LIN {X 104.168,Y 46.841,Z 66.500,A 180.000,B 0.000,C 180.000} C_DIS
LIN {X 104.160,Y 46.662,Z 66.500,A 180.000,B 0.000,C 180.000} C_DIS
LIN {X 104.143,Y 46.483,Z 66.500,A 180.000,B 0.000,C 180.000} C_DIS
LIN {X 104.121,Y 46.275,Z 66.500,A 180.000,B 0.000,C 180.000} C_DIS
LIN {X 104.105,Y 46.126,Z 66.500,A 180.000,B 0.000,C 180.000} C_DIS
LIN {X 104.086,Y 45.947,Z 66.500,A 180.000,B 0.000,C 180.000} C_DIS
LIN {X 104.059,Y 45.768,Z 66.500,A 180.000,B 0.000,C 180.000} C_DIS
LIN {X 103.998,Y 45.411,Z 66.500,A 180.000,B 0.000,C 180.000} C_DIS
LIN {X 103.967,Y 45.232,Z 66.500,A 180.000,B 0.000,C 180.000} C_DIS
LIN {X 103.929,Y 45.053,Z 66.500,A 180.000,B 0.000,C 180.000} C_DIS
LIN {X 103.845,Y 44.696,Z 66.500,A 180.000,B 0.000,C 180.000} C_DIS
LIN {X 103.802,Y 44.517,Z 66.500,A 180.000,B 0.000,C 180.000} C_DIS
LIN {X 103.752,Y 44.338,Z 66.500,A 180.000,B 0.000,C 180.000} C_DIS
LIN {X 103.644,Y 43.981,Z 66.500,A 180.000,B 0.000,C 180.000} C_DIS
LIN {X 103.589,Y 43.802,Z 66.500,A 180.000,B 0.000,C 180.000} C_DIS
LIN {X 103.526,Y 43.623,Z 66.500,A 180.000,B 0.000,C 180.000} C_DIS
LIN {X 103.392,Y 43.266,Z 66.500,A 180.000,B 0.000,C 180.000} C_DIS
LIN {X 103.332,Y 43.106,Z 66.500,A 180.000,B 0.000,C 180.000} C_DIS
LIN {X 103.325,Y 43.087,Z 66.500,A 180.000,B 0.000,C 180.000} C_DIS
LIN {X 103.247,Y 42.908,Z 66.500,A 180.000,B 0.000,C 180.000} C_DIS
LIN {X 103.087,Y 42.550,Z 66.500,A 180.000,B 0.000,C 180.000} C_DIS
LIN {X 103.005,Y 42.372,Z 66.500,A 180.000,B 0.000,C 180.000} C_DIS
LIN {X 102.975,Y 42.314,Z 66.500,A 180.000,B 0.000,C 180.000} C_DIS
LIN {X 102.724,Y 41.835,Z 66.500,A 180.000,B 0.000,C 180.000} C_DIS
LIN {X 102.623,Y 41.657,Z 66.500,A 180.000,B 0.000,C 180.000} C_DIS
LIN {X 102.406,Y 41.299,Z 66.500,A 180.000,B 0.000,C 180.000} C_DIS
LIN {X 102.296,Y 41.120,Z 66.500,A 180.000,B 0.000,C 180.000} C_DIS
LIN {X 102.260,Y 41.067,Z 66.500,A 180.000,B 0.000,C 180.000} C_DIS
LIN {X 102.172,Y 40.942,Z 66.500,A 180.000,B 0.000,C 180.000} C_DIS
LIN {X 101.923,Y 40.584,Z 66.500,A 180.000,B 0.000,C 180.000} C_DIS
LIN {X 101.902,Y 40.554,Z 66.500,A 180.000,B 0.000,C 180.000} C_DIS
LIN {X 101.788,Y 40.405,Z 66.500,A 180.000,B 0.000,C 180.000} C_DIS
LIN {X 101.504,Y 40.048,Z 66.500,A 180.000,B 0.000,C 180.000} C_DIS
LIN {X 101.366,Y 39.883,Z 66.500,A 180.000,B 0.000,C 180.000} C_DIS
LIN {X 101.008,Y 39.486,Z 66.500,A 180.000,B 0.000,C 180.000} C_DIS
LIN {X 100.861,Y 39.333,Z 66.500,A 180.000,B 0.000,C 180.000} C_DIS
LIN {X 100.472,Y 38.952,Z 66.500,A 180.000,B 0.000,C 180.000} C_DIS
LIN {X 100.300,Y 38.796,Z 66.500,A 180.000,B 0.000,C 180.000} C_DIS
LIN {X 99.936,Y 38.482,Z 66.500,A 180.000,B 0.000,C 180.000} C_DIS
LIN {X 99.885,Y 38.439,Z 66.500,A 180.000,B 0.000,C 180.000} C_DIS
LIN {X 99.757,Y 38.338,Z 66.500,A 180.000,B 0.000,C 180.000} C_DIS
LIN {X 99.399,Y 38.067,Z 66.500,A 180.000,B 0.000,C 180.000} C_DIS
LIN {X 99.221,Y 37.936,Z 66.500,A 180.000,B 0.000,C 180.000} C_DIS
LIN {X 99.171,Y 37.902,Z 66.500,A 180.000,B 0.000,C 180.000} C_DIS
LIN {X 98.863,Y 37.698,Z 66.500,A 180.000,B 0.000,C 180.000} C_DIS
LIN {X 98.684,Y 37.580,Z 66.500,A 180.000,B 0.000,C 180.000} C_DIS
LIN {X 98.627,Y 37.545,Z 66.500,A 180.000,B 0.000,C 180.000} C_DIS
LIN {X 98.505,Y 37.474,Z 66.500,A 180.000,B 0.000,C 180.000} C_DIS
LIN {X 98.148,Y 37.268,Z 66.500,A 180.000,B 0.000,C 180.000} C_DIS
LIN {X 98.005,Y 37.187,Z 66.500,A 180.000,B 0.000,C 180.000} C_DIS
LIN {X 97.969,Y 37.169,Z 66.500,A 180.000,B 0.000,C 180.000} C_DIS
LIN {X 97.790,Y 37.080,Z 66.500,A 180.000,B 0.000,C 180.000} C_DIS
LIN {X 97.433,Y 36.903,Z 66.500,A 180.000,B 0.000,C 180.000} C_DIS
LIN {X 97.272,Y 36.830,Z 66.500,A 180.000,B 0.000,C 180.000} C_DIS
LIN {X 96.846,Y 36.651,Z 66.500,A 180.000,B 0.000,C 180.000} C_DIS
LIN {X 96.718,Y 36.598,Z 66.500,A 180.000,B 0.000,C 180.000} C_DIS
LIN {X 96.539,Y 36.533,Z 66.500,A 180.000,B 0.000,C 180.000} C_DIS
LIN {X 96.181,Y 36.409,Z 66.500,A 180.000,B 0.000,C 180.000} C_DIS
LIN {X 96.003,Y 36.347,Z 66.500,A 180.000,B 0.000,C 180.000} C_DIS
LIN {X 95.824,Y 36.296,Z 66.500,A 180.000,B 0.000,C 180.000} C_DIS
LIN {X 95.466,Y 36.196,Z 66.500,A 180.000,B 0.000,C 180.000} C_DIS
LIN {X 95.288,Y 36.147,Z 66.500,A 180.000,B 0.000,C 180.000} C_DIS
LIN {X 95.141,Y 36.115,Z 66.500,A 180.000,B 0.000,C 180.000} C_DIS
LIN {X 94.751,Y 36.032,Z 66.500,A 180.000,B 0.000,C 180.000} C_DIS
LIN {X 94.573,Y 35.995,Z 66.500,A 180.000,B 0.000,C 180.000} C_DIS
LIN {X 94.394,Y 35.967,Z 66.500,A 180.000,B 0.000,C 180.000} C_DIS
LIN {X 94.036,Y 35.915,Z 66.500,A 180.000,B 0.000,C 180.000} C_DIS
LIN {X 93.857,Y 35.889,Z 66.500,A 180.000,B 0.000,C 180.000} C_DIS
LIN {X 93.679,Y 35.872,Z 66.500,A 180.000,B 0.000,C 180.000} C_DIS
LIN {X 93.321,Y 35.843,Z 66.500,A 180.000,B 0.000,C 180.000} C_DIS
LIN {X 93.142,Y 35.828,Z 66.500,A 180.000,B 0.000,C 180.000} C_DIS
LIN {X 92.964,Y 35.822,Z 66.500,A 180.000,B 0.000,C 180.000} C_DIS
LIN {X 92.606,Y 35.814,Z 66.500,A 180.000,B 0.000,C 180.000} C_DIS
LIN {X 92.427,Y 35.811,Z 66.500,A 180.000,B 0.000,C 180.000} C_DIS
LIN {X 92.249,Y 35.815,Z 66.500,A 180.000,B 0.000,C 180.000} C_DIS
LIN {X 91.712,Y 35.838,Z 66.500,A 180.000,B 0.000,C 180.000} C_DIS
LIN {X 91.533,Y 35.852,Z 66.500,A 180.000,B 0.000,C 180.000} C_DIS
LIN {X 90.997,Y 35.908,Z 66.500,A 180.000,B 0.000,C 180.000} C_DIS
LIN {X 90.872,Y 35.926,Z 66.500,A 180.000,B 0.000,C 180.000} C_DIS
; Link Move Starts
LIN {X 90.783,Y 35.936,Z 66.500,A 180.000,B 0.000,C 180.000} C_DIS
LIN {X 90.702,Y 35.950,Z 66.500,A 180.000,B 0.000,C 180.000} C_DIS
LIN {X 90.699,Y 35.950,Z 66.500,A 180.000,B 0.000,C 180.000} C_DIS
LIN {X 90.693,Y 35.947,Z 66.500,A 180.000,B 0.000,C 180.000} C_DIS
LIN {X 90.541,Y 35.852,Z 66.500,A 180.000,B 0.000,C 180.000} C_DIS
LIN {X 90.371,Y 35.764,Z 66.499,A 180.000,B 0.000,C 180.000} C_DIS
LIN {X 90.194,Y 35.689,Z 66.499,A 180.000,B 0.000,C 180.000} C_DIS
LIN {X 90.035,Y 35.634,Z 66.498,A 180.000,B 0.000,C 180.000} C_DIS
LIN {X 89.873,Y 35.590,Z 66.497,A 180.000,B 0.000,C 180.000} C_DIS
LIN {X 89.718,Y 35.559,Z 66.496,A 180.000,B 0.000,C 180.000} C_DIS
LIN {X 89.562,Y 35.538,Z 66.495,A 180.000,B 0.000,C 180.000} C_DIS
LIN {X 89.405,Y 35.527,Z 66.494,A 180.000,B 0.000,C 180.000} C_DIS
LIN {X 89.247,Y 35.525,Z 66.493,A 180.000,B 0.000,C 180.000} C_DIS
LIN {X 89.090,Y 35.534,Z 66.492,A 180.000,B 0.000,C 180.000} C_DIS
LIN {X 88.934,Y 35.552,Z 66.490,A 180.000,B 0.000,C 180.000} C_DIS
LIN {X 88.779,Y 35.580,Z 66.489,A 180.000,B 0.000,C 180.000} C_DIS
LIN {X 88.626,Y 35.618,Z 66.487,A 180.000,B 0.000,C 180.000} C_DIS
LIN {X 88.326,Y 35.716,Z 66.483,A 180.000,B 0.000,C 180.000} C_DIS
LIN {X 88.028,Y 35.817,Z 66.479,A 180.000,B 0.000,C 180.000} C_DIS
LIN {X 87.730,Y 35.917,Z 66.475,A 180.000,B 0.000,C 180.000} C_DIS
LIN {X 87.431,Y 36.018,Z 66.470,A 180.000,B 0.000,C 180.000} C_DIS
LIN {X 87.282,Y 36.068,Z 66.467,A 180.000,B 0.000,C 180.000} C_DIS
LIN {X 87.133,Y 36.119,Z 66.465,A 180.000,B 0.000,C 180.000} C_DIS
LIN {X 86.983,Y 36.169,Z 66.462,A 180.000,B 0.000,C 180.000} C_DIS
LIN {X 86.834,Y 36.219,Z 66.459,A 180.000,B 0.000,C 180.000} C_DIS
LIN {X 86.685,Y 36.270,Z 66.456,A 180.000,B 0.000,C 180.000} C_DIS
LIN {X 86.536,Y 36.320,Z 66.453,A 180.000,B 0.000,C 180.000} C_DIS
LIN {X 86.386,Y 36.370,Z 66.450,A 180.000,B 0.000,C 180.000} C_DIS
LIN {X 86.237,Y 36.421,Z 66.446,A 180.000,B 0.000,C 180.000} C_DIS
LIN {X 86.088,Y 36.471,Z 66.443,A 180.000,B 0.000,C 180.000} C_DIS
LIN {X 85.939,Y 36.521,Z 66.440,A 180.000,B 0.000,C 180.000} C_DIS
LIN {X 85.789,Y 36.572,Z 66.436,A 180.000,B 0.000,C 180.000} C_DIS
LIN {X 85.640,Y 36.622,Z 66.433,A 180.000,B 0.000,C 180.000} C_DIS
LIN {X 85.491,Y 36.672,Z 66.429,A 180.000,B 0.000,C 180.000} C_DIS
LIN {X 85.342,Y 36.723,Z 66.425,A 180.000,B 0.000,C 180.000} C_DIS
LIN {X 85.193,Y 36.773,Z 66.421,A 180.000,B 0.000,C 180.000} C_DIS
LIN {X 85.043,Y 36.823,Z 66.417,A 180.000,B 0.000,C 180.000} C_DIS
LIN {X 84.894,Y 36.874,Z 66.413,A 180.000,B 0.000,C 180.000} C_DIS
LIN {X 84.745,Y 36.924,Z 66.409,A 180.000,B 0.000,C 180.000} C_DIS
LIN {X 84.596,Y 36.974,Z 66.405,A 180.000,B 0.000,C 180.000} C_DIS
LIN {X 84.446,Y 37.025,Z 66.401,A 180.000,B 0.000,C 180.000} C_DIS
LIN {X 84.297,Y 37.075,Z 66.397,A 180.000,B 0.000,C 180.000} C_DIS
LIN {X 84.148,Y 37.125,Z 66.392,A 180.000,B 0.000,C 180.000} C_DIS
LIN {X 83.999,Y 37.176,Z 66.388,A 180.000,B 0.000,C 180.000} C_DIS
LIN {X 83.849,Y 37.226,Z 66.383,A 180.000,B 0.000,C 180.000} C_DIS
LIN {X 83.700,Y 37.277,Z 66.379,A 180.000,B 0.000,C 180.000} C_DIS
LIN {X 83.551,Y 37.327,Z 66.374,A 180.000,B 0.000,C 180.000} C_DIS
LIN {X 83.402,Y 37.377,Z 66.369,A 180.000,B 0.000,C 180.000} C_DIS
LIN {X 83.252,Y 37.428,Z 66.364,A 180.000,B 0.000,C 180.000} C_DIS
LIN {X 83.103,Y 37.478,Z 66.359,A 180.000,B 0.000,C 180.000} C_DIS
LIN {X 82.954,Y 37.528,Z 66.355,A 180.000,B 0.000,C 180.000} C_DIS
LIN {X 82.879,Y 37.553,Z 66.352,A 180.000,B 0.000,C 180.000} C_DIS
LIN {X 82.805,Y 37.579,Z 66.350,A 180.000,B 0.000,C 180.000} C_DIS
LIN {X 82.730,Y 37.604,Z 66.347,A 180.000,B 0.000,C 180.000} C_DIS
LIN {X 82.655,Y 37.629,Z 66.344,A 180.000,B 0.000,C 180.000} C_DIS
LIN {X 82.581,Y 37.654,Z 66.342,A 180.000,B 0.000,C 180.000} C_DIS
LIN {X 82.506,Y 37.679,Z 66.339,A 180.000,B 0.000,C 180.000} C_DIS
LIN {X 82.432,Y 37.704,Z 66.337,A 180.000,B 0.000,C 180.000} C_DIS
LIN {X 82.282,Y 37.755,Z 66.332,A 180.000,B 0.000,C 180.000} C_DIS
LIN {X 82.133,Y 37.805,Z 66.326,A 180.000,B 0.000,C 180.000} C_DIS
LIN {X 81.984,Y 37.855,Z 66.321,A 180.000,B 0.000,C 180.000} C_DIS
LIN {X 81.835,Y 37.906,Z 66.315,A 180.000,B 0.000,C 180.000} C_DIS
LIN {X 81.685,Y 37.956,Z 66.310,A 180.000,B 0.000,C 180.000} C_DIS
LIN {X 81.536,Y 38.007,Z 66.305,A 180.000,B 0.000,C 180.000} C_DIS
LIN {X 81.462,Y 38.032,Z 66.302,A 180.000,B 0.000,C 180.000} C_DIS
LIN {X 81.312,Y 38.082,Z 66.296,A 180.000,B 0.000,C 180.000} C_DIS
LIN {X 81.089,Y 38.158,Z 66.288,A 180.000,B 0.000,C 180.000} C_DIS
LIN {X 80.939,Y 38.208,Z 66.283,A 180.000,B 0.000,C 180.000} C_DIS
LIN {X 80.865,Y 38.233,Z 66.280,A 180.000,B 0.000,C 180.000} C_DIS
LIN {X 80.715,Y 38.283,Z 66.274,A 180.000,B 0.000,C 180.000} C_DIS
LIN {X 80.492,Y 38.359,Z 66.266,A 180.000,B 0.000,C 180.000} C_DIS
LIN {X 80.342,Y 38.409,Z 66.261,A 180.000,B 0.000,C 180.000} C_DIS
LIN {X 80.268,Y 38.434,Z 66.258,A 180.000,B 0.000,C 180.000} C_DIS
LIN {X 80.118,Y 38.485,Z 66.252,A 180.000,B 0.000,C 180.000} C_DIS
LIN {X 79.895,Y 38.560,Z 66.244,A 180.000,B 0.000,C 180.000} C_DIS
LIN {X 79.745,Y 38.611,Z 66.239,A 180.000,B 0.000,C 180.000} C_DIS
LIN {X 79.671,Y 38.636,Z 66.236,A 180.000,B 0.000,C 180.000} C_DIS
LIN {X 79.522,Y 38.686,Z 66.230,A 180.000,B 0.000,C 180.000} C_DIS
LIN {X 79.223,Y 38.787,Z 66.219,A 180.000,B 0.000,C 180.000} C_DIS
LIN {X 78.775,Y 38.938,Z 66.203,A 180.000,B 0.000,C 180.000} C_DIS
LIN {X 78.626,Y 38.988,Z 66.197,A 180.000,B 0.000,C 180.000} C_DIS
LIN {X 78.178,Y 39.139,Z 66.181,A 180.000,B 0.000,C 180.000} C_DIS
LIN {X 78.029,Y 39.190,Z 66.175,A 180.000,B 0.000,C 180.000} C_DIS
LIN {X 77.581,Y 39.341,Z 66.159,A 180.000,B 0.000,C 180.000} C_DIS
LIN {X 77.358,Y 39.416,Z 66.151,A 180.000,B 0.000,C 180.000} C_DIS
LIN {X 77.208,Y 39.467,Z 66.145,A 180.000,B 0.000,C 180.000} C_DIS
LIN {X 76.761,Y 39.618,Z 66.129,A 180.000,B 0.000,C 180.000} C_DIS
LIN {X 76.611,Y 39.668,Z 66.123,A 180.000,B 0.000,C 180.000} C_DIS
LIN {X 76.164,Y 39.819,Z 66.107,A 180.000,B 0.000,C 180.000} C_DIS
LIN {X 75.940,Y 39.894,Z 66.098,A 180.000,B 0.000,C 180.000} C_DIS
LIN {X 75.119,Y 40.171,Z 66.068,A 180.000,B 0.000,C 180.000} C_DIS
LIN {X 74.074,Y 40.524,Z 66.030,A 180.000,B 0.000,C 180.000} C_DIS
LIN {X 73.179,Y 40.826,Z 65.997,A 180.000,B 0.000,C 180.000} C_DIS
LIN {X 64.822,Y 43.645,Z 65.689,A 180.000,B 0.000,C 180.000} C_DIS
LIN {X 64.673,Y 43.695,Z 65.683,A 180.000,B 0.000,C 180.000} C_DIS
LIN {X 64.523,Y 43.746,Z 65.678,A 180.000,B 0.000,C 180.000} C_DIS
LIN {X 64.374,Y 43.796,Z 65.672,A 180.000,B 0.000,C 180.000} C_DIS
LIN {X 64.225,Y 43.847,Z 65.667,A 180.000,B 0.000,C 180.000} C_DIS
LIN {X 64.150,Y 43.872,Z 65.664,A 180.000,B 0.000,C 180.000} C_DIS
LIN {X 64.076,Y 43.897,Z 65.662,A 180.000,B 0.000,C 180.000} C_DIS
LIN {X 64.001,Y 43.922,Z 65.659,A 180.000,B 0.000,C 180.000} C_DIS
LIN {X 63.926,Y 43.947,Z 65.657,A 180.000,B 0.000,C 180.000} C_DIS
LIN {X 63.852,Y 43.972,Z 65.654,A 180.000,B 0.000,C 180.000} C_DIS
LIN {X 63.777,Y 43.998,Z 65.652,A 180.000,B 0.000,C 180.000} C_DIS
LIN {X 63.702,Y 44.023,Z 65.649,A 180.000,B 0.000,C 180.000} C_DIS
LIN {X 63.553,Y 44.073,Z 65.644,A 180.000,B 0.000,C 180.000} C_DIS
LIN {X 63.404,Y 44.123,Z 65.639,A 180.000,B 0.000,C 180.000} C_DIS
LIN {X 63.255,Y 44.174,Z 65.634,A 180.000,B 0.000,C 180.000} C_DIS
LIN {X 63.106,Y 44.224,Z 65.630,A 180.000,B 0.000,C 180.000} C_DIS
LIN {X 62.956,Y 44.274,Z 65.625,A 180.000,B 0.000,C 180.000} C_DIS
LIN {X 62.807,Y 44.325,Z 65.620,A 180.000,B 0.000,C 180.000} C_DIS
LIN {X 62.658,Y 44.375,Z 65.616,A 180.000,B 0.000,C 180.000} C_DIS
LIN {X 62.509,Y 44.425,Z 65.611,A 180.000,B 0.000,C 180.000} C_DIS
LIN {X 62.359,Y 44.476,Z 65.607,A 180.000,B 0.000,C 180.000} C_DIS
LIN {X 62.210,Y 44.526,Z 65.602,A 180.000,B 0.000,C 180.000} C_DIS
LIN {X 62.061,Y 44.576,Z 65.598,A 180.000,B 0.000,C 180.000} C_DIS
LIN {X 61.912,Y 44.627,Z 65.594,A 180.000,B 0.000,C 180.000} C_DIS
LIN {X 61.762,Y 44.677,Z 65.590,A 180.000,B 0.000,C 180.000} C_DIS
LIN {X 61.613,Y 44.728,Z 65.586,A 180.000,B 0.000,C 180.000} C_DIS
LIN {X 61.464,Y 44.778,Z 65.582,A 180.000,B 0.000,C 180.000} C_DIS
LIN {X 61.315,Y 44.828,Z 65.578,A 180.000,B 0.000,C 180.000} C_DIS
LIN {X 61.165,Y 44.879,Z 65.574,A 180.000,B 0.000,C 180.000} C_DIS
LIN {X 61.016,Y 44.929,Z 65.570,A 180.000,B 0.000,C 180.000} C_DIS
LIN {X 60.867,Y 44.979,Z 65.566,A 180.000,B 0.000,C 180.000} C_DIS
LIN {X 60.718,Y 45.030,Z 65.563,A 180.000,B 0.000,C 180.000} C_DIS
LIN {X 60.569,Y 45.080,Z 65.559,A 180.000,B 0.000,C 180.000} C_DIS
LIN {X 60.419,Y 45.130,Z 65.556,A 180.000,B 0.000,C 180.000} C_DIS
LIN {X 60.270,Y 45.181,Z 65.553,A 180.000,B 0.000,C 180.000} C_DIS
LIN {X 60.121,Y 45.231,Z 65.549,A 180.000,B 0.000,C 180.000} C_DIS
LIN {X 59.972,Y 45.281,Z 65.546,A 180.000,B 0.000,C 180.000} C_DIS
LIN {X 59.822,Y 45.332,Z 65.543,A 180.000,B 0.000,C 180.000} C_DIS
LIN {X 59.673,Y 45.382,Z 65.540,A 180.000,B 0.000,C 180.000} C_DIS
LIN {X 59.524,Y 45.432,Z 65.537,A 180.000,B 0.000,C 180.000} C_DIS
LIN {X 59.375,Y 45.483,Z 65.535,A 180.000,B 0.000,C 180.000} C_DIS
LIN {X 59.225,Y 45.533,Z 65.532,A 180.000,B 0.000,C 180.000} C_DIS
LIN {X 59.076,Y 45.583,Z 65.529,A 180.000,B 0.000,C 180.000} C_DIS
LIN {X 58.778,Y 45.684,Z 65.525,A 180.000,B 0.000,C 180.000} C_DIS
LIN {X 58.479,Y 45.785,Z 65.520,A 180.000,B 0.000,C 180.000} C_DIS
LIN {X 58.181,Y 45.885,Z 65.516,A 180.000,B 0.000,C 180.000} C_DIS
LIN {X 57.882,Y 45.986,Z 65.513,A 180.000,B 0.000,C 180.000} C_DIS
LIN {X 57.584,Y 46.087,Z 65.509,A 180.000,B 0.000,C 180.000} C_DIS
LIN {X 57.285,Y 46.188,Z 65.507,A 180.000,B 0.000,C 180.000} C_DIS
LIN {X 56.987,Y 46.288,Z 65.504,A 180.000,B 0.000,C 180.000} C_DIS
LIN {X 56.688,Y 46.389,Z 65.503,A 180.000,B 0.000,C 180.000} C_DIS
LIN {X 56.390,Y 46.490,Z 65.501,A 180.000,B 0.000,C 180.000} C_DIS
LIN {X 56.091,Y 46.590,Z 65.500,A 180.000,B 0.000,C 180.000} C_DIS
LIN {X 55.793,Y 46.691,Z 65.500,A 180.000,B 0.000,C 180.000} C_DIS
LIN {X 55.704,Y 46.721,Z 65.500,A 180.000,B 0.000,C 180.000} C_DIS
; Cutting Move Starts
LIN {X 45.590,Y 50.133,Z 65.500,A 180.000,B 0.000,C 180.000} C_DIS
LIN {X 45.411,Y 50.194,Z 65.500,A 180.000,B 0.000,C 180.000} C_DIS
LIN {X 45.296,Y 50.238,Z 65.500,A 180.000,B 0.000,C 180.000} C_DIS
LIN {X 45.232,Y 50.265,Z 65.500,A 180.000,B 0.000,C 180.000} C_DIS
LIN {X 45.053,Y 50.353,Z 65.500,A 180.000,B 0.000,C 180.000} C_DIS
LIN {X 44.944,Y 50.416,Z 65.500,A 180.000,B 0.000,C 180.000} C_DIS
LIN {X 44.874,Y 50.461,Z 65.500,A 180.000,B 0.000,C 180.000} C_DIS
LIN {X 44.785,Y 50.522,Z 65.500,A 180.000,B 0.000,C 180.000} C_DIS
LIN {X 44.696,Y 50.590,Z 65.500,A 180.000,B 0.000,C 180.000} C_DIS
LIN {X 44.689,Y 50.595,Z 65.500,A 180.000,B 0.000,C 180.000} C_DIS
LIN {X 44.603,Y 50.667,Z 65.500,A 180.000,B 0.000,C 180.000} C_DIS
LIN {X 44.517,Y 50.746,Z 65.500,A 180.000,B 0.000,C 180.000} C_DIS
LIN {X 44.488,Y 50.774,Z 65.500,A 180.000,B 0.000,C 180.000} C_DIS
LIN {X 44.410,Y 50.855,Z 65.500,A 180.000,B 0.000,C 180.000} C_DIS
LIN {X 44.338,Y 50.936,Z 65.500,A 180.000,B 0.000,C 180.000} C_DIS
LIN {X 44.325,Y 50.953,Z 65.500,A 180.000,B 0.000,C 180.000} C_DIS
LIN {X 44.254,Y 51.042,Z 65.500,A 180.000,B 0.000,C 180.000} C_DIS
LIN {X 44.189,Y 51.131,Z 65.500,A 180.000,B 0.000,C 180.000} C_DIS
LIN {X 44.159,Y 51.176,Z 65.500,A 180.000,B 0.000,C 180.000} C_DIS
LIN {X 44.077,Y 51.310,Z 65.500,A 180.000,B 0.000,C 180.000} C_DIS
LIN {X 43.984,Y 51.489,Z 65.500,A 180.000,B 0.000,C 180.000} C_DIS
LIN {X 43.981,Y 51.497,Z 65.500,A 180.000,B 0.000,C 180.000} C_DIS
LIN {X 43.909,Y 51.668,Z 65.500,A 180.000,B 0.000,C 180.000} C_DIS
LIN {X 43.849,Y 51.847,Z 65.500,A 180.000,B 0.000,C 180.000} C_DIS
LIN {X 43.804,Y 52.025,Z 65.500,A 180.000,B 0.000,C 180.000} C_DIS
LIN {X 43.802,Y 52.035,Z 65.500,A 180.000,B 0.000,C 180.000} C_DIS
LIN {X 43.772,Y 52.204,Z 65.500,A 180.000,B 0.000,C 180.000} C_DIS
LIN {X 43.754,Y 52.383,Z 65.500,A 180.000,B 0.000,C 180.000} C_DIS
LIN {X 43.748,Y 52.562,Z 65.500,A 180.000,B 0.000,C 180.000} C_DIS
LIN {X 43.756,Y 52.740,Z 65.500,A 180.000,B 0.000,C 180.000} C_DIS
LIN {X 43.776,Y 52.919,Z 65.500,A 180.000,B 0.000,C 180.000} C_DIS
LIN {X 43.802,Y 53.064,Z 65.500,A 180.000,B 0.000,C 180.000} C_DIS
LIN {X 43.809,Y 53.098,Z 65.500,A 180.000,B 0.000,C 180.000} C_DIS
LIN {X 43.856,Y 53.277,Z 65.500,A 180.000,B 0.000,C 180.000} C_DIS
LIN {X 43.916,Y 53.455,Z 65.500,A 180.000,B 0.000,C 180.000} C_DIS
LIN {X 50.248,Y 72.226,Z 65.500,A 180.000,B 0.000,C 180.000} C_DIS
LIN {X 50.311,Y 72.405,Z 65.500,A 180.000,B 0.000,C 180.000} C_DIS
LIN {X 50.388,Y 72.584,Z 65.500,A 180.000,B 0.000,C 180.000} C_DIS
LIN {X 50.416,Y 72.640,Z 65.500,A 180.000,B 0.000,C 180.000} C_DIS
LIN {X 50.484,Y 72.763,Z 65.500,A 180.000,B 0.000,C 180.000} C_DIS
LIN {X 50.595,Y 72.936,Z 65.500,A 180.000,B 0.000,C 180.000} C_DIS
LIN {X 50.599,Y 72.941,Z 65.500,A 180.000,B 0.000,C 180.000} C_DIS
LIN {X 50.665,Y 73.031,Z 65.500,A 180.000,B 0.000,C 180.000} C_DIS
LIN {X 50.737,Y 73.120,Z 65.500,A 180.000,B 0.000,C 180.000} C_DIS
LIN {X 50.774,Y 73.162,Z 65.500,A 180.000,B 0.000,C 180.000} C_DIS
LIN {X 50.905,Y 73.299,Z 65.500,A 180.000,B 0.000,C 180.000} C_DIS
LIN {X 50.953,Y 73.343,Z 65.500,A 180.000,B 0.000,C 180.000} C_DIS
LIN {X 51.112,Y 73.478,Z 65.500,A 180.000,B 0.000,C 180.000} C_DIS
LIN {X 51.131,Y 73.493,Z 65.500,A 180.000,B 0.000,C 180.000} C_DIS
LIN {X 51.310,Y 73.616,Z 65.500,A 180.000,B 0.000,C 180.000} C_DIS
LIN {X 51.376,Y 73.656,Z 65.500,A 180.000,B 0.000,C 180.000} C_DIS
LIN {X 51.489,Y 73.719,Z 65.500,A 180.000,B 0.000,C 180.000} C_DIS
LIN {X 51.668,Y 73.803,Z 65.500,A 180.000,B 0.000,C 180.000} C_DIS
LIN {X 51.749,Y 73.835,Z 65.500,A 180.000,B 0.000,C 180.000} C_DIS
LIN {X 51.847,Y 73.870,Z 65.500,A 180.000,B 0.000,C 180.000} C_DIS
LIN {X 52.025,Y 73.923,Z 65.500,A 180.000,B 0.000,C 180.000} C_DIS
LIN {X 52.204,Y 73.961,Z 65.500,A 180.000,B 0.000,C 180.000} C_DIS
LIN {X 52.383,Y 73.987,Z 65.500,A 180.000,B 0.000,C 180.000} C_DIS
LIN {X 52.562,Y 73.999,Z 65.500,A 180.000,B 0.000,C 180.000} C_DIS
LIN {X 52.740,Y 73.998,Z 65.500,A 180.000,B 0.000,C 180.000} C_DIS
LIN {X 52.919,Y 73.985,Z 65.500,A 180.000,B 0.000,C 180.000} C_DIS
LIN {X 53.098,Y 73.958,Z 65.500,A 180.000,B 0.000,C 180.000} C_DIS
LIN {X 53.277,Y 73.918,Z 65.500,A 180.000,B 0.000,C 180.000} C_DIS
LIN {X 53.455,Y 73.864,Z 65.500,A 180.000,B 0.000,C 180.000} C_DIS
LIN {X 83.198,Y 63.830,Z 65.500,A 180.000,B 0.000,C 180.000} C_DIS
LIN {X 96.464,Y 59.355,Z 65.500,A 180.000,B 0.000,C 180.000} C_DIS
LIN {X 96.539,Y 59.329,Z 65.500,A 180.000,B 0.000,C 180.000} C_DIS
LIN {X 96.718,Y 59.257,Z 65.500,A 180.000,B 0.000,C 180.000} C_DIS
LIN {X 96.883,Y 59.176,Z 65.500,A 180.000,B 0.000,C 180.000} C_DIS
LIN {X 96.897,Y 59.169,Z 65.500,A 180.000,B 0.000,C 180.000} C_DIS
LIN {X 97.075,Y 59.061,Z 65.500,A 180.000,B 0.000,C 180.000} C_DIS
LIN {X 97.167,Y 58.997,Z 65.500,A 180.000,B 0.000,C 180.000} C_DIS
LIN {X 97.254,Y 58.931,Z 65.500,A 180.000,B 0.000,C 180.000} C_DIS
LIN {X 97.385,Y 58.819,Z 65.500,A 180.000,B 0.000,C 180.000} C_DIS
LIN {X 97.433,Y 58.774,Z 65.500,A 180.000,B 0.000,C 180.000} C_DIS
LIN {X 97.562,Y 58.640,Z 65.500,A 180.000,B 0.000,C 180.000} C_DIS
LIN {X 97.612,Y 58.582,Z 65.500,A 180.000,B 0.000,C 180.000} C_DIS
LIN {X 97.707,Y 58.461,Z 65.500,A 180.000,B 0.000,C 180.000} C_DIS
LIN {X 97.716,Y 58.449,Z 65.500,A 180.000,B 0.000,C 180.000} C_DIS
LIN {X 97.722,Y 58.440,Z 65.500,A 180.000,B 0.000,C 180.000} C_DIS
LIN {X 97.724,Y 58.438,Z 65.500,A 180.000,B 0.000,C 180.000} C_DIS
LIN {X 97.728,Y 58.437,Z 65.500,A 180.000,B 0.000,C 180.000} C_DIS
LIN {X 97.749,Y 58.427,Z 65.500,A 180.000,B 0.000,C 180.000} C_DIS
LIN {X 97.790,Y 58.407,Z 65.500,A 180.000,B 0.000,C 180.000} C_DIS
LIN {X 97.969,Y 58.315,Z 65.500,A 180.000,B 0.000,C 180.000} C_DIS
LIN {X 98.373,Y 58.103,Z 65.500,A 180.000,B 0.000,C 180.000} C_DIS
LIN {X 98.505,Y 58.030,Z 65.500,A 180.000,B 0.000,C 180.000} C_DIS
LIN {X 98.684,Y 57.922,Z 65.500,A 180.000,B 0.000,C 180.000} C_DIS
LIN {X 99.042,Y 57.705,Z 65.500,A 180.000,B 0.000,C 180.000} C_DIS
LIN {X 99.221,Y 57.586,Z 65.500,A 180.000,B 0.000,C 180.000} C_DIS
LIN {X 99.578,Y 57.337,Z 65.500,A 180.000,B 0.000,C 180.000} C_DIS
LIN {X 99.757,Y 57.210,Z 65.500,A 180.000,B 0.000,C 180.000} C_DIS
LIN {X 99.758,Y 57.210,Z 65.500,A 180.000,B 0.000,C 180.000} C_DIS
LIN {X 99.936,Y 57.069,Z 65.500,A 180.000,B 0.000,C 180.000} C_DIS
LIN {X 100.209,Y 56.852,Z 65.500,A 180.000,B 0.000,C 180.000} C_DIS
LIN {X 100.293,Y 56.785,Z 65.500,A 180.000,B 0.000,C 180.000} C_DIS
LIN {X 100.422,Y 56.673,Z 65.500,A 180.000,B 0.000,C 180.000} C_DIS
LIN {X 100.829,Y 56.306,Z 65.500,A 180.000,B 0.000,C 180.000} C_DIS
LIN {X 101.003,Y 56.137,Z 65.500,A 180.000,B 0.000,C 180.000} C_DIS
LIN {X 101.366,Y 55.766,Z 65.500,A 180.000,B 0.000,C 180.000} C_DIS
LIN {X 101.516,Y 55.601,Z 65.500,A 180.000,B 0.000,C 180.000} C_DIS
LIN {X 101.824,Y 55.243,Z 65.500,A 180.000,B 0.000,C 180.000} C_DIS
LIN {X 101.902,Y 55.152,Z 65.500,A 180.000,B 0.000,C 180.000} C_DIS
LIN {X 101.972,Y 55.064,Z 65.500,A 180.000,B 0.000,C 180.000} C_DIS
LIN {X 102.260,Y 54.685,Z 65.500,A 180.000,B 0.000,C 180.000} C_DIS
LIN {X 102.377,Y 54.528,Z 65.500,A 180.000,B 0.000,C 180.000} C_DIS
LIN {X 102.438,Y 54.439,Z 65.500,A 180.000,B 0.000,C 180.000} C_DIS
LIN {X 102.735,Y 53.992,Z 65.500,A 180.000,B 0.000,C 180.000} C_DIS
LIN {X 102.796,Y 53.899,Z 65.500,A 180.000,B 0.000,C 180.000} C_DIS
LIN {X 102.848,Y 53.813,Z 65.500,A 180.000,B 0.000,C 180.000} C_DIS
LIN {X 103.054,Y 53.455,Z 65.500,A 180.000,B 0.000,C 180.000} C_DIS
LIN {X 103.153,Y 53.283,Z 65.500,A 180.000,B 0.000,C 180.000} C_DIS
LIN {X 103.157,Y 53.277,Z 65.500,A 180.000,B 0.000,C 180.000} C_DIS
LIN {X 103.250,Y 53.098,Z 65.500,A 180.000,B 0.000,C 180.000} C_DIS
LIN {X 103.427,Y 52.740,Z 65.500,A 180.000,B 0.000,C 180.000} C_DIS
LIN {X 103.511,Y 52.570,Z 65.500,A 180.000,B 0.000,C 180.000} C_DIS
LIN {X 103.515,Y 52.562,Z 65.500,A 180.000,B 0.000,C 180.000} C_DIS
LIN {X 103.592,Y 52.383,Z 65.500,A 180.000,B 0.000,C 180.000} C_DIS
LIN {X 103.742,Y 52.025,Z 65.500,A 180.000,B 0.000,C 180.000} C_DIS
LIN {X 103.816,Y 51.847,Z 65.500,A 180.000,B 0.000,C 180.000} C_DIS
LIN {X 103.869,Y 51.701,Z 65.500,A 180.000,B 0.000,C 180.000} C_DIS
LIN {X 104.047,Y 51.187,Z 65.500,A 180.000,B 0.000,C 180.000} C_DIS
LIN {X 104.066,Y 51.131,Z 65.500,A 180.000,B 0.000,C 180.000} C_DIS
LIN {X 104.117,Y 50.953,Z 65.500,A 180.000,B 0.000,C 180.000} C_DIS
LIN {X 104.226,Y 50.562,Z 65.500,A 180.000,B 0.000,C 180.000} C_DIS
LIN {X 104.266,Y 50.416,Z 65.500,A 180.000,B 0.000,C 180.000} C_DIS
LIN {X 104.307,Y 50.238,Z 65.500,A 180.000,B 0.000,C 180.000} C_DIS
LIN {X 104.405,Y 49.774,Z 65.500,A 180.000,B 0.000,C 180.000} C_DIS
LIN {X 104.420,Y 49.701,Z 65.500,A 180.000,B 0.000,C 180.000} C_DIS
LIN {X 104.451,Y 49.523,Z 65.500,A 180.000,B 0.000,C 180.000} C_DIS
LIN {X 104.529,Y 48.986,Z 65.500,A 180.000,B 0.000,C 180.000} C_DIS
LIN {X 104.551,Y 48.807,Z 65.500,A 180.000,B 0.000,C 180.000} C_DIS
LIN {X 104.595,Y 48.271,Z 65.500,A 180.000,B 0.000,C 180.000} C_DIS
LIN {X 104.608,Y 48.092,Z 65.500,A 180.000,B 0.000,C 180.000} C_DIS
LIN {X 104.612,Y 47.914,Z 65.500,A 180.000,B 0.000,C 180.000} C_DIS
LIN {X 104.619,Y 47.556,Z 65.500,A 180.000,B 0.000,C 180.000} C_DIS
LIN {X 104.622,Y 47.377,Z 65.500,A 180.000,B 0.000,C 180.000} C_DIS
LIN {X 104.616,Y 47.198,Z 65.500,A 180.000,B 0.000,C 180.000} C_DIS
LIN {X 104.601,Y 46.841,Z 65.500,A 180.000,B 0.000,C 180.000} C_DIS
LIN {X 104.593,Y 46.662,Z 65.500,A 180.000,B 0.000,C 180.000} C_DIS
LIN {X 104.584,Y 46.539,Z 65.500,A 180.000,B 0.000,C 180.000} C_DIS
LIN {X 104.578,Y 46.483,Z 65.500,A 180.000,B 0.000,C 180.000} C_DIS
LIN {X 104.521,Y 45.947,Z 65.500,A 180.000,B 0.000,C 180.000} C_DIS
LIN {X 104.497,Y 45.768,Z 65.500,A 180.000,B 0.000,C 180.000} C_DIS
LIN {X 104.405,Y 45.225,Z 65.500,A 180.000,B 0.000,C 180.000} C_DIS
LIN {X 104.373,Y 45.053,Z 65.500,A 180.000,B 0.000,C 180.000} C_DIS
LIN {X 104.331,Y 44.874,Z 65.500,A 180.000,B 0.000,C 180.000} C_DIS
LIN {X 104.226,Y 44.429,Z 65.500,A 180.000,B 0.000,C 180.000} C_DIS
LIN {X 104.203,Y 44.338,Z 65.500,A 180.000,B 0.000,C 180.000} C_DIS
LIN {X 104.150,Y 44.159,Z 65.500,A 180.000,B 0.000,C 180.000} C_DIS
LIN {X 104.041,Y 43.802,Z 65.500,A 180.000,B 0.000,C 180.000} C_DIS
LIN {X 103.986,Y 43.623,Z 65.500,A 180.000,B 0.000,C 180.000} C_DIS
LIN {X 103.920,Y 43.444,Z 65.500,A 180.000,B 0.000,C 180.000} C_DIS
LIN {X 103.787,Y 43.087,Z 65.500,A 180.000,B 0.000,C 180.000} C_DIS
LIN {X 103.719,Y 42.908,Z 65.500,A 180.000,B 0.000,C 180.000} C_DIS
LIN {X 103.690,Y 42.840,Z 65.500,A 180.000,B 0.000,C 180.000} C_DIS
LIN {X 103.481,Y 42.372,Z 65.500,A 180.000,B 0.000,C 180.000} C_DIS
LIN {X 103.399,Y 42.193,Z 65.500,A 180.000,B 0.000,C 180.000} C_DIS
LIN {X 103.332,Y 42.064,Z 65.500,A 180.000,B 0.000,C 180.000} C_DIS
LIN {X 103.119,Y 41.657,Z 65.500,A 180.000,B 0.000,C 180.000} C_DIS
LIN {X 103.020,Y 41.478,Z 65.500,A 180.000,B 0.000,C 180.000} C_DIS
LIN {X 102.796,Y 41.109,Z 65.500,A 180.000,B 0.000,C 180.000} C_DIS
LIN {X 102.694,Y 40.942,Z 65.500,A 180.000,B 0.000,C 180.000} C_DIS
LIN {X 102.617,Y 40.824,Z 65.500,A 180.000,B 0.000,C 180.000} C_DIS
LIN {X 102.326,Y 40.405,Z 65.500,A 180.000,B 0.000,C 180.000} C_DIS
LIN {X 102.260,Y 40.310,Z 65.500,A 180.000,B 0.000,C 180.000} C_DIS
LIN {X 102.197,Y 40.226,Z 65.500,A 180.000,B 0.000,C 180.000} C_DIS
LIN {X 102.081,Y 40.079,Z 65.500,A 180.000,B 0.000,C 180.000} C_DIS
LIN {X 101.902,Y 39.854,Z 65.500,A 180.000,B 0.000,C 180.000} C_DIS
LIN {X 101.771,Y 39.690,Z 65.500,A 180.000,B 0.000,C 180.000} C_DIS
LIN {X 101.723,Y 39.634,Z 65.500,A 180.000,B 0.000,C 180.000} C_DIS
LIN {X 101.613,Y 39.511,Z 65.500,A 180.000,B 0.000,C 180.000} C_DIS
LIN {X 101.366,Y 39.237,Z 65.500,A 180.000,B 0.000,C 180.000} C_DIS
LIN {X 101.291,Y 39.154,Z 65.500,A 180.000,B 0.000,C 180.000} C_DIS
LIN {X 101.187,Y 39.046,Z 65.500,A 180.000,B 0.000,C 180.000} C_DIS
LIN {X 100.829,Y 38.697,Z 65.500,A 180.000,B 0.000,C 180.000} C_DIS
LIN {X 100.749,Y 38.618,Z 65.500,A 180.000,B 0.000,C 180.000} C_DIS
LIN {X 100.651,Y 38.528,Z 65.500,A 180.000,B 0.000,C 180.000} C_DIS
LIN {X 100.548,Y 38.439,Z 65.500,A 180.000,B 0.000,C 180.000} C_DIS
LIN {X 100.293,Y 38.219,Z 65.500,A 180.000,B 0.000,C 180.000} C_DIS
LIN {X 100.132,Y 38.081,Z 65.500,A 180.000,B 0.000,C 180.000} C_DIS
LIN {X 100.114,Y 38.067,Z 65.500,A 180.000,B 0.000,C 180.000} C_DIS
LIN {X 99.936,Y 37.931,Z 65.500,A 180.000,B 0.000,C 180.000} C_DIS
LIN {X 99.578,Y 37.660,Z 65.500,A 180.000,B 0.000,C 180.000} C_DIS
LIN {X 99.414,Y 37.545,Z 65.500,A 180.000,B 0.000,C 180.000} C_DIS
LIN {X 99.042,Y 37.298,Z 65.500,A 180.000,B 0.000,C 180.000} C_DIS
LIN {X 98.872,Y 37.187,Z 65.500,A 180.000,B 0.000,C 180.000} C_DIS
LIN {X 98.863,Y 37.182,Z 65.500,A 180.000,B 0.000,C 180.000} C_DIS
LIN {X 98.684,Y 37.078,Z 65.500,A 180.000,B 0.000,C 180.000} C_DIS
LIN {X 98.327,Y 36.872,Z 65.500,A 180.000,B 0.000,C 180.000} C_DIS
LIN {X 98.253,Y 36.830,Z 65.500,A 180.000,B 0.000,C 180.000} C_DIS
LIN {X 98.148,Y 36.775,Z 65.500,A 180.000,B 0.000,C 180.000} C_DIS
LIN {X 97.612,Y 36.509,Z 65.500,A 180.000,B 0.000,C 180.000} C_DIS
LIN {X 97.534,Y 36.472,Z 65.500,A 180.000,B 0.000,C 180.000} C_DIS
LIN {X 97.433,Y 36.429,Z 65.500,A 180.000,B 0.000,C 180.000} C_DIS
LIN {X 97.075,Y 36.279,Z 65.500,A 180.000,B 0.000,C 180.000} C_DIS
LIN {X 96.897,Y 36.204,Z 65.500,A 180.000,B 0.000,C 180.000} C_DIS
LIN {X 96.718,Y 36.137,Z 65.500,A 180.000,B 0.000,C 180.000} C_DIS
LIN {X 96.360,Y 36.013,Z 65.500,A 180.000,B 0.000,C 180.000} C_DIS
LIN {X 96.181,Y 35.951,Z 65.500,A 180.000,B 0.000,C 180.000} C_DIS
LIN {X 96.137,Y 35.936,Z 65.500,A 180.000,B 0.000,C 180.000} C_DIS
LIN {X 96.003,Y 35.897,Z 65.500,A 180.000,B 0.000,C 180.000} C_DIS
LIN {X 95.466,Y 35.747,Z 65.500,A 180.000,B 0.000,C 180.000} C_DIS
LIN {X 95.288,Y 35.704,Z 65.500,A 180.000,B 0.000,C 180.000} C_DIS
LIN {X 94.751,Y 35.590,Z 65.500,A 180.000,B 0.000,C 180.000} C_DIS
LIN {X 94.695,Y 35.578,Z 65.500,A 180.000,B 0.000,C 180.000} C_DIS
LIN {X 94.573,Y 35.557,Z 65.500,A 180.000,B 0.000,C 180.000} C_DIS
LIN {X 94.394,Y 35.530,Z 65.500,A 180.000,B 0.000,C 180.000} C_DIS
LIN {X 94.036,Y 35.478,Z 65.500,A 180.000,B 0.000,C 180.000} C_DIS
LIN {X 93.857,Y 35.454,Z 65.500,A 180.000,B 0.000,C 180.000} C_DIS
LIN {X 93.679,Y 35.438,Z 65.500,A 180.000,B 0.000,C 180.000} C_DIS
LIN {X 93.213,Y 35.400,Z 65.500,A 180.000,B 0.000,C 180.000} C_DIS
LIN {X 93.142,Y 35.395,Z 65.500,A 180.000,B 0.000,C 180.000} C_DIS
LIN {X 92.964,Y 35.389,Z 65.500,A 180.000,B 0.000,C 180.000} C_DIS
LIN {X 92.606,Y 35.382,Z 65.500,A 180.000,B 0.000,C 180.000} C_DIS
LIN {X 92.427,Y 35.378,Z 65.500,A 180.000,B 0.000,C 180.000} C_DIS
LIN {X 92.249,Y 35.382,Z 65.500,A 180.000,B 0.000,C 180.000} C_DIS
LIN {X 91.712,Y 35.405,Z 65.500,A 180.000,B 0.000,C 180.000} C_DIS
LIN {X 91.533,Y 35.417,Z 65.500,A 180.000,B 0.000,C 180.000} C_DIS
LIN {X 91.355,Y 35.436,Z 65.500,A 180.000,B 0.000,C 180.000} C_DIS
LIN {X 90.997,Y 35.474,Z 65.500,A 180.000,B 0.000,C 180.000} C_DIS
LIN {X 90.818,Y 35.495,Z 65.500,A 180.000,B 0.000,C 180.000} C_DIS
LIN {X 90.640,Y 35.525,Z 65.500,A 180.000,B 0.000,C 180.000} C_DIS
LIN {X 90.282,Y 35.585,Z 65.500,A 180.000,B 0.000,C 180.000} C_DIS
LIN {X 90.103,Y 35.617,Z 65.500,A 180.000,B 0.000,C 180.000} C_DIS
LIN {X 90.059,Y 35.626,Z 65.500,A 180.000,B 0.000,C 180.000} C_DIS
LIN {X 90.036,Y 35.631,Z 65.500,A 180.000,B 0.000,C 180.000} C_DIS
LIN {X 90.031,Y 35.632,Z 65.500,A 180.000,B 0.000,C 180.000} C_DIS
LIN {X 90.029,Y 35.632,Z 65.500,A 180.000,B 0.000,C 180.000} C_DIS
LIN {X 90.025,Y 35.631,Z 65.500,A 180.000,B 0.000,C 180.000} C_DIS
LIN {X 90.014,Y 35.628,Z 65.500,A 180.000,B 0.000,C 180.000} C_DIS
LIN {X 89.925,Y 35.603,Z 65.500,A 180.000,B 0.000,C 180.000} C_DIS
LIN {X 89.819,Y 35.578,Z 65.500,A 180.000,B 0.000,C 180.000} C_DIS
LIN {X 89.746,Y 35.564,Z 65.500,A 180.000,B 0.000,C 180.000} C_DIS
LIN {X 89.567,Y 35.539,Z 65.500,A 180.000,B 0.000,C 180.000} C_DIS
LIN {X 89.388,Y 35.526,Z 65.500,A 180.000,B 0.000,C 180.000} C_DIS
LIN {X 89.209,Y 35.526,Z 65.500,A 180.000,B 0.000,C 180.000} C_DIS
LIN {X 89.031,Y 35.540,Z 65.500,A 180.000,B 0.000,C 180.000} C_DIS
LIN {X 88.852,Y 35.566,Z 65.500,A 180.000,B 0.000,C 180.000} C_DIS
LIN {X 88.788,Y 35.578,Z 65.500,A 180.000,B 0.000,C 180.000} C_DIS
LIN {X 88.673,Y 35.605,Z 65.500,A 180.000,B 0.000,C 180.000} C_DIS
LIN {X 88.494,Y 35.659,Z 65.500,A 180.000,B 0.000,C 180.000} C_DIS
LIN {X 55.704,Y 46.721,Z 65.500,A 180.000,B 0.000,C 180.000} C_DIS
; Link Move Starts
LIN {X 55.405,Y 46.822,Z 65.500,A 180.000,B 0.000,C 180.000} C_DIS
LIN {X 55.107,Y 46.922,Z 65.499,A 180.000,B 0.000,C 180.000} C_DIS
LIN {X 54.808,Y 47.023,Z 65.498,A 180.000,B 0.000,C 180.000} C_DIS
LIN {X 54.510,Y 47.124,Z 65.496,A 180.000,B 0.000,C 180.000} C_DIS
LIN {X 54.211,Y 47.225,Z 65.494,A 180.000,B 0.000,C 180.000} C_DIS
LIN {X 53.913,Y 47.325,Z 65.491,A 180.000,B 0.000,C 180.000} C_DIS
LIN {X 53.614,Y 47.426,Z 65.488,A 180.000,B 0.000,C 180.000} C_DIS
LIN {X 53.316,Y 47.527,Z 65.485,A 180.000,B 0.000,C 180.000} C_DIS
LIN {X 53.017,Y 47.627,Z 65.481,A 180.000,B 0.000,C 180.000} C_DIS
LIN {X 52.719,Y 47.728,Z 65.477,A 180.000,B 0.000,C 180.000} C_DIS
LIN {X 52.421,Y 47.829,Z 65.472,A 180.000,B 0.000,C 180.000} C_DIS
LIN {X 52.271,Y 47.879,Z 65.469,A 180.000,B 0.000,C 180.000} C_DIS
LIN {X 52.122,Y 47.929,Z 65.467,A 180.000,B 0.000,C 180.000} C_DIS
LIN {X 51.973,Y 47.980,Z 65.464,A 180.000,B 0.000,C 180.000} C_DIS
LIN {X 51.824,Y 48.030,Z 65.461,A 180.000,B 0.000,C 180.000} C_DIS
LIN {X 51.674,Y 48.080,Z 65.459,A 180.000,B 0.000,C 180.000} C_DIS
LIN {X 51.525,Y 48.131,Z 65.456,A 180.000,B 0.000,C 180.000} C_DIS
LIN {X 51.376,Y 48.181,Z 65.452,A 180.000,B 0.000,C 180.000} C_DIS
LIN {X 51.227,Y 48.231,Z 65.449,A 180.000,B 0.000,C 180.000} C_DIS
LIN {X 51.077,Y 48.282,Z 65.446,A 180.000,B 0.000,C 180.000} C_DIS
LIN {X 50.928,Y 48.332,Z 65.443,A 180.000,B 0.000,C 180.000} C_DIS
LIN {X 50.779,Y 48.382,Z 65.439,A 180.000,B 0.000,C 180.000} C_DIS
LIN {X 50.630,Y 48.433,Z 65.436,A 180.000,B 0.000,C 180.000} C_DIS
LIN {X 50.480,Y 48.483,Z 65.432,A 180.000,B 0.000,C 180.000} C_DIS
LIN {X 50.331,Y 48.534,Z 65.428,A 180.000,B 0.000,C 180.000} C_DIS
LIN {X 50.182,Y 48.584,Z 65.425,A 180.000,B 0.000,C 180.000} C_DIS
LIN {X 50.033,Y 48.634,Z 65.421,A 180.000,B 0.000,C 180.000} C_DIS
LIN {X 49.883,Y 48.685,Z 65.417,A 180.000,B 0.000,C 180.000} C_DIS
LIN {X 49.734,Y 48.735,Z 65.413,A 180.000,B 0.000,C 180.000} C_DIS
LIN {X 49.585,Y 48.785,Z 65.409,A 180.000,B 0.000,C 180.000} C_DIS
LIN {X 49.436,Y 48.836,Z 65.405,A 180.000,B 0.000,C 180.000} C_DIS
LIN {X 49.287,Y 48.886,Z 65.400,A 180.000,B 0.000,C 180.000} C_DIS
LIN {X 49.137,Y 48.936,Z 65.396,A 180.000,B 0.000,C 180.000} C_DIS
LIN {X 48.988,Y 48.987,Z 65.392,A 180.000,B 0.000,C 180.000} C_DIS
LIN {X 48.839,Y 49.037,Z 65.387,A 180.000,B 0.000,C 180.000} C_DIS
LIN {X 48.690,Y 49.087,Z 65.383,A 180.000,B 0.000,C 180.000} C_DIS
LIN {X 48.540,Y 49.138,Z 65.378,A 180.000,B 0.000,C 180.000} C_DIS
LIN {X 48.391,Y 49.188,Z 65.373,A 180.000,B 0.000,C 180.000} C_DIS
LIN {X 48.242,Y 49.238,Z 65.369,A 180.000,B 0.000,C 180.000} C_DIS
LIN {X 48.093,Y 49.289,Z 65.364,A 180.000,B 0.000,C 180.000} C_DIS
LIN {X 47.943,Y 49.339,Z 65.359,A 180.000,B 0.000,C 180.000} C_DIS
LIN {X 47.794,Y 49.389,Z 65.354,A 180.000,B 0.000,C 180.000} C_DIS
LIN {X 47.720,Y 49.415,Z 65.351,A 180.000,B 0.000,C 180.000} C_DIS
LIN {X 47.645,Y 49.440,Z 65.349,A 180.000,B 0.000,C 180.000} C_DIS
LIN {X 47.570,Y 49.465,Z 65.346,A 180.000,B 0.000,C 180.000} C_DIS
LIN {X 47.496,Y 49.490,Z 65.344,A 180.000,B 0.000,C 180.000} C_DIS
LIN {X 47.421,Y 49.515,Z 65.341,A 180.000,B 0.000,C 180.000} C_DIS
LIN {X 47.346,Y 49.540,Z 65.339,A 180.000,B 0.000,C 180.000} C_DIS
LIN {X 47.272,Y 49.566,Z 65.336,A 180.000,B 0.000,C 180.000} C_DIS
LIN {X 47.123,Y 49.616,Z 65.331,A 180.000,B 0.000,C 180.000} C_DIS
LIN {X 46.973,Y 49.666,Z 65.325,A 180.000,B 0.000,C 180.000} C_DIS
LIN {X 46.824,Y 49.717,Z 65.320,A 180.000,B 0.000,C 180.000} C_DIS
LIN {X 46.675,Y 49.767,Z 65.315,A 180.000,B 0.000,C 180.000} C_DIS
LIN {X 46.526,Y 49.817,Z 65.309,A 180.000,B 0.000,C 180.000} C_DIS
LIN {X 46.451,Y 49.842,Z 65.307,A 180.000,B 0.000,C 180.000} C_DIS
LIN {X 46.302,Y 49.893,Z 65.301,A 180.000,B 0.000,C 180.000} C_DIS
LIN {X 46.078,Y 49.968,Z 65.293,A 180.000,B 0.000,C 180.000} C_DIS
LIN {X 45.929,Y 50.019,Z 65.287,A 180.000,B 0.000,C 180.000} C_DIS
LIN {X 45.854,Y 50.044,Z 65.285,A 180.000,B 0.000,C 180.000} C_DIS
LIN {X 45.705,Y 50.094,Z 65.279,A 180.000,B 0.000,C 180.000} C_DIS
LIN {X 45.481,Y 50.170,Z 65.271,A 180.000,B 0.000,C 180.000} C_DIS
LIN {X 45.407,Y 50.195,Z 65.268,A 180.000,B 0.000,C 180.000} C_DIS
LIN {X 45.333,Y 50.223,Z 65.265,A 180.000,B 0.000,C 180.000} C_DIS
LIN {X 45.260,Y 50.253,Z 65.263,A 180.000,B 0.000,C 180.000} C_DIS
LIN {X 45.188,Y 50.285,Z 65.260,A 180.000,B 0.000,C 180.000} C_DIS
LIN {X 45.117,Y 50.320,Z 65.257,A 180.000,B 0.000,C 180.000} C_DIS
LIN {X 45.048,Y 50.356,Z 65.254,A 180.000,B 0.000,C 180.000} C_DIS
LIN {X 44.979,Y 50.395,Z 65.252,A 180.000,B 0.000,C 180.000} C_DIS
LIN {X 44.912,Y 50.436,Z 65.249,A 180.000,B 0.000,C 180.000} C_DIS
LIN {X 44.846,Y 50.480,Z 65.246,A 180.000,B 0.000,C 180.000} C_DIS
LIN {X 44.782,Y 50.525,Z 65.243,A 180.000,B 0.000,C 180.000} C_DIS
LIN {X 44.719,Y 50.572,Z 65.241,A 180.000,B 0.000,C 180.000} C_DIS
LIN {X 44.657,Y 50.621,Z 65.238,A 180.000,B 0.000,C 180.000} C_DIS
LIN {X 44.597,Y 50.672,Z 65.235,A 180.000,B 0.000,C 180.000} C_DIS
LIN {X 44.539,Y 50.725,Z 65.232,A 180.000,B 0.000,C 180.000} C_DIS
LIN {X 44.482,Y 50.780,Z 65.230,A 180.000,B 0.000,C 180.000} C_DIS
LIN {X 44.427,Y 50.836,Z 65.227,A 180.000,B 0.000,C 180.000} C_DIS
LIN {X 44.374,Y 50.895,Z 65.224,A 180.000,B 0.000,C 180.000} C_DIS
LIN {X 44.323,Y 50.954,Z 65.221,A 180.000,B 0.000,C 180.000} C_DIS
LIN {X 44.274,Y 51.016,Z 65.219,A 180.000,B 0.000,C 180.000} C_DIS
LIN {X 44.226,Y 51.079,Z 65.216,A 180.000,B 0.000,C 180.000} C_DIS
LIN {X 44.181,Y 51.143,Z 65.213,A 180.000,B 0.000,C 180.000} C_DIS
LIN {X 44.138,Y 51.209,Z 65.210,A 180.000,B 0.000,C 180.000} C_DIS
LIN {X 44.097,Y 51.276,Z 65.208,A 180.000,B 0.000,C 180.000} C_DIS
LIN {X 44.058,Y 51.345,Z 65.205,A 180.000,B 0.000,C 180.000} C_DIS
LIN {X 44.021,Y 51.414,Z 65.202,A 180.000,B 0.000,C 180.000} C_DIS
LIN {X 43.986,Y 51.485,Z 65.199,A 180.000,B 0.000,C 180.000} C_DIS
LIN {X 43.954,Y 51.557,Z 65.197,A 180.000,B 0.000,C 180.000} C_DIS
LIN {X 43.924,Y 51.629,Z 65.194,A 180.000,B 0.000,C 180.000} C_DIS
LIN {X 43.896,Y 51.703,Z 65.191,A 180.000,B 0.000,C 180.000} C_DIS
LIN {X 43.870,Y 51.778,Z 65.188,A 180.000,B 0.000,C 180.000} C_DIS
LIN {X 43.847,Y 51.853,Z 65.186,A 180.000,B 0.000,C 180.000} C_DIS
LIN {X 43.826,Y 51.929,Z 65.183,A 180.000,B 0.000,C 180.000} C_DIS
LIN {X 43.808,Y 52.006,Z 65.180,A 180.000,B 0.000,C 180.000} C_DIS
LIN {X 43.792,Y 52.083,Z 65.177,A 180.000,B 0.000,C 180.000} C_DIS
LIN {X 43.779,Y 52.160,Z 65.175,A 180.000,B 0.000,C 180.000} C_DIS
LIN {X 43.768,Y 52.238,Z 65.172,A 180.000,B 0.000,C 180.000} C_DIS
LIN {X 43.759,Y 52.317,Z 65.169,A 180.000,B 0.000,C 180.000} C_DIS
LIN {X 43.753,Y 52.395,Z 65.166,A 180.000,B 0.000,C 180.000} C_DIS
LIN {X 43.749,Y 52.474,Z 65.164,A 180.000,B 0.000,C 180.000} C_DIS
LIN {X 43.748,Y 52.553,Z 65.161,A 180.000,B 0.000,C 180.000} C_DIS
LIN {X 43.750,Y 52.631,Z 65.158,A 180.000,B 0.000,C 180.000} C_DIS
LIN {X 43.753,Y 52.710,Z 65.155,A 180.000,B 0.000,C 180.000} C_DIS
LIN {X 43.760,Y 52.789,Z 65.153,A 180.000,B 0.000,C 180.000} C_DIS
LIN {X 43.769,Y 52.867,Z 65.150,A 180.000,B 0.000,C 180.000} C_DIS
LIN {X 43.780,Y 52.945,Z 65.147,A 180.000,B 0.000,C 180.000} C_DIS
LIN {X 43.793,Y 53.022,Z 65.144,A 180.000,B 0.000,C 180.000} C_DIS
LIN {X 43.810,Y 53.099,Z 65.142,A 180.000,B 0.000,C 180.000} C_DIS
LIN {X 43.828,Y 53.176,Z 65.139,A 180.000,B 0.000,C 180.000} C_DIS
LIN {X 43.849,Y 53.252,Z 65.136,A 180.000,B 0.000,C 180.000} C_DIS
LIN {X 43.872,Y 53.327,Z 65.133,A 180.000,B 0.000,C 180.000} C_DIS
LIN {X 43.897,Y 53.402,Z 65.131,A 180.000,B 0.000,C 180.000} C_DIS
LIN {X 43.973,Y 53.626,Z 65.122,A 180.000,B 0.000,C 180.000} C_DIS
LIN {X 44.023,Y 53.775,Z 65.117,A 180.000,B 0.000,C 180.000} C_DIS
LIN {X 44.174,Y 54.223,Z 65.100,A 180.000,B 0.000,C 180.000} C_DIS
LIN {X 44.250,Y 54.446,Z 65.092,A 180.000,B 0.000,C 180.000} C_DIS
LIN {X 44.602,Y 55.491,Z 65.054,A 180.000,B 0.000,C 180.000} C_DIS
LIN {X 44.778,Y 56.013,Z 65.034,A 180.000,B 0.000,C 180.000} C_DIS
LIN {X 45.030,Y 56.760,Z 65.007,A 180.000,B 0.000,C 180.000} C_DIS
LIN {X 46.893,Y 62.281,Z 64.803,A 180.000,B 0.000,C 180.000} C_DIS
LIN {X 46.918,Y 62.356,Z 64.801,A 180.000,B 0.000,C 180.000} C_DIS
LIN {X 46.968,Y 62.505,Z 64.795,A 180.000,B 0.000,C 180.000} C_DIS
LIN {X 47.120,Y 62.953,Z 64.779,A 180.000,B 0.000,C 180.000} C_DIS
LIN {X 47.170,Y 63.102,Z 64.773,A 180.000,B 0.000,C 180.000} C_DIS
LIN {X 47.245,Y 63.326,Z 64.765,A 180.000,B 0.000,C 180.000} C_DIS
LIN {X 47.296,Y 63.475,Z 64.759,A 180.000,B 0.000,C 180.000} C_DIS
LIN {X 47.321,Y 63.550,Z 64.757,A 180.000,B 0.000,C 180.000} C_DIS
LIN {X 47.371,Y 63.699,Z 64.751,A 180.000,B 0.000,C 180.000} C_DIS
LIN {X 47.447,Y 63.923,Z 64.743,A 180.000,B 0.000,C 180.000} C_DIS
LIN {X 47.497,Y 64.072,Z 64.737,A 180.000,B 0.000,C 180.000} C_DIS
LIN {X 47.522,Y 64.147,Z 64.735,A 180.000,B 0.000,C 180.000} C_DIS
LIN {X 47.573,Y 64.296,Z 64.729,A 180.000,B 0.000,C 180.000} C_DIS
LIN {X 47.648,Y 64.520,Z 64.721,A 180.000,B 0.000,C 180.000} C_DIS
LIN {X 47.698,Y 64.669,Z 64.715,A 180.000,B 0.000,C 180.000} C_DIS
LIN {X 47.724,Y 64.744,Z 64.713,A 180.000,B 0.000,C 180.000} C_DIS
LIN {X 47.774,Y 64.893,Z 64.707,A 180.000,B 0.000,C 180.000} C_DIS
LIN {X 47.850,Y 65.117,Z 64.699,A 180.000,B 0.000,C 180.000} C_DIS
LIN {X 47.900,Y 65.266,Z 64.693,A 180.000,B 0.000,C 180.000} C_DIS
LIN {X 48.001,Y 65.564,Z 64.682,A 180.000,B 0.000,C 180.000} C_DIS
LIN {X 48.051,Y 65.714,Z 64.677,A 180.000,B 0.000,C 180.000} C_DIS
LIN {X 48.101,Y 65.863,Z 64.672,A 180.000,B 0.000,C 180.000} C_DIS
LIN {X 48.152,Y 66.012,Z 64.666,A 180.000,B 0.000,C 180.000} C_DIS
LIN {X 48.177,Y 66.087,Z 64.664,A 180.000,B 0.000,C 180.000} C_DIS
LIN {X 48.202,Y 66.161,Z 64.661,A 180.000,B 0.000,C 180.000} C_DIS
LIN {X 48.227,Y 66.236,Z 64.659,A 180.000,B 0.000,C 180.000} C_DIS
LIN {X 48.252,Y 66.311,Z 64.656,A 180.000,B 0.000,C 180.000} C_DIS
LIN {X 48.277,Y 66.385,Z 64.654,A 180.000,B 0.000,C 180.000} C_DIS
LIN {X 48.303,Y 66.460,Z 64.651,A 180.000,B 0.000,C 180.000} C_DIS
LIN {X 48.328,Y 66.535,Z 64.649,A 180.000,B 0.000,C 180.000} C_DIS
LIN {X 48.378,Y 66.684,Z 64.644,A 180.000,B 0.000,C 180.000} C_DIS
LIN {X 48.428,Y 66.833,Z 64.639,A 180.000,B 0.000,C 180.000} C_DIS
LIN {X 48.479,Y 66.982,Z 64.634,A 180.000,B 0.000,C 180.000} C_DIS
LIN {X 48.529,Y 67.131,Z 64.629,A 180.000,B 0.000,C 180.000} C_DIS
LIN {X 48.580,Y 67.281,Z 64.624,A 180.000,B 0.000,C 180.000} C_DIS
LIN {X 48.630,Y 67.430,Z 64.620,A 180.000,B 0.000,C 180.000} C_DIS
LIN {X 48.680,Y 67.579,Z 64.615,A 180.000,B 0.000,C 180.000} C_DIS
LIN {X 48.731,Y 67.728,Z 64.611,A 180.000,B 0.000,C 180.000} C_DIS
LIN {X 48.781,Y 67.878,Z 64.606,A 180.000,B 0.000,C 180.000} C_DIS
LIN {X 48.831,Y 68.027,Z 64.602,A 180.000,B 0.000,C 180.000} C_DIS
LIN {X 48.882,Y 68.176,Z 64.597,A 180.000,B 0.000,C 180.000} C_DIS
LIN {X 48.932,Y 68.325,Z 64.593,A 180.000,B 0.000,C 180.000} C_DIS
LIN {X 48.982,Y 68.475,Z 64.589,A 180.000,B 0.000,C 180.000} C_DIS
LIN {X 49.033,Y 68.624,Z 64.585,A 180.000,B 0.000,C 180.000} C_DIS
LIN {X 49.083,Y 68.773,Z 64.581,A 180.000,B 0.000,C 180.000} C_DIS
LIN {X 49.133,Y 68.922,Z 64.577,A 180.000,B 0.000,C 180.000} C_DIS
LIN {X 49.184,Y 69.072,Z 64.573,A 180.000,B 0.000,C 180.000} C_DIS
LIN {X 49.234,Y 69.221,Z 64.570,A 180.000,B 0.000,C 180.000} C_DIS
LIN {X 49.284,Y 69.370,Z 64.566,A 180.000,B 0.000,C 180.000} C_DIS
LIN {X 49.335,Y 69.519,Z 64.562,A 180.000,B 0.000,C 180.000} C_DIS
LIN {X 49.385,Y 69.668,Z 64.559,A 180.000,B 0.000,C 180.000} C_DIS
LIN {X 49.435,Y 69.818,Z 64.556,A 180.000,B 0.000,C 180.000} C_DIS
LIN {X 49.486,Y 69.967,Z 64.552,A 180.000,B 0.000,C 180.000} C_DIS
LIN {X 49.536,Y 70.116,Z 64.549,A 180.000,B 0.000,C 180.000} C_DIS
LIN {X 49.586,Y 70.265,Z 64.546,A 180.000,B 0.000,C 180.000} C_DIS
LIN {X 49.637,Y 70.415,Z 64.543,A 180.000,B 0.000,C 180.000} C_DIS
LIN {X 49.687,Y 70.564,Z 64.540,A 180.000,B 0.000,C 180.000} C_DIS
LIN {X 49.737,Y 70.713,Z 64.537,A 180.000,B 0.000,C 180.000} C_DIS
LIN {X 49.788,Y 70.862,Z 64.534,A 180.000,B 0.000,C 180.000} C_DIS
LIN {X 49.838,Y 71.012,Z 64.532,A 180.000,B 0.000,C 180.000} C_DIS
LIN {X 49.888,Y 71.161,Z 64.529,A 180.000,B 0.000,C 180.000} C_DIS
LIN {X 49.939,Y 71.310,Z 64.527,A 180.000,B 0.000,C 180.000} C_DIS
LIN {X 50.040,Y 71.609,Z 64.522,A 180.000,B 0.000,C 180.000} C_DIS
LIN {X 50.140,Y 71.907,Z 64.518,A 180.000,B 0.000,C 180.000} C_DIS
LIN {X 50.241,Y 72.206,Z 64.514,A 180.000,B 0.000,C 180.000} C_DIS
LIN {X 50.292,Y 72.355,Z 64.512,A 180.000,B 0.000,C 180.000} C_DIS
LIN {X 50.350,Y 72.501,Z 64.511,A 180.000,B 0.000,C 180.000} C_DIS
LIN {X 50.418,Y 72.643,Z 64.509,A 180.000,B 0.000,C 180.000} C_DIS
LIN {X 50.494,Y 72.781,Z 64.508,A 180.000,B 0.000,C 180.000} C_DIS
LIN {X 50.579,Y 72.913,Z 64.507,A 180.000,B 0.000,C 180.000} C_DIS
LIN {X 50.672,Y 73.040,Z 64.505,A 180.000,B 0.000,C 180.000} C_DIS
LIN {X 50.773,Y 73.161,Z 64.504,A 180.000,B 0.000,C 180.000} C_DIS
LIN {X 50.882,Y 73.276,Z 64.503,A 180.000,B 0.000,C 180.000} C_DIS
LIN {X 50.997,Y 73.383,Z 64.503,A 180.000,B 0.000,C 180.000} C_DIS
LIN {X 51.119,Y 73.483,Z 64.502,A 180.000,B 0.000,C 180.000} C_DIS
LIN {X 51.247,Y 73.575,Z 64.501,A 180.000,B 0.000,C 180.000} C_DIS
LIN {X 51.380,Y 73.659,Z 64.501,A 180.000,B 0.000,C 180.000} C_DIS
LIN {X 51.518,Y 73.734,Z 64.500,A 180.000,B 0.000,C 180.000} C_DIS
LIN {X 51.661,Y 73.800,Z 64.500,A 180.000,B 0.000,C 180.000} C_DIS
LIN {X 51.769,Y 73.843,Z 64.500,A 180.000,B 0.000,C 180.000} C_DIS
LIN {X 51.880,Y 73.880,Z 64.500,A 180.000,B 0.000,C 180.000} C_DIS
; Cutting Move Starts
LIN {X 52.025,Y 73.923,Z 64.500,A 180.000,B 0.000,C 180.000} C_DIS
LIN {X 52.204,Y 73.961,Z 64.500,A 180.000,B 0.000,C 180.000} C_DIS
LIN {X 52.383,Y 73.987,Z 64.500,A 180.000,B 0.000,C 180.000} C_DIS
LIN {X 52.562,Y 73.999,Z 64.500,A 180.000,B 0.000,C 180.000} C_DIS
LIN {X 52.740,Y 73.998,Z 64.500,A 180.000,B 0.000,C 180.000} C_DIS
LIN {X 52.919,Y 73.985,Z 64.500,A 180.000,B 0.000,C 180.000} C_DIS
LIN {X 53.098,Y 73.958,Z 64.500,A 180.000,B 0.000,C 180.000} C_DIS
LIN {X 53.277,Y 73.918,Z 64.500,A 180.000,B 0.000,C 180.000} C_DIS
LIN {X 53.455,Y 73.864,Z 64.500,A 180.000,B 0.000,C 180.000} C_DIS
LIN {X 83.198,Y 63.830,Z 64.500,A 180.000,B 0.000,C 180.000} C_DIS
LIN {X 96.464,Y 59.355,Z 64.500,A 180.000,B 0.000,C 180.000} C_DIS
LIN {X 96.539,Y 59.329,Z 64.500,A 180.000,B 0.000,C 180.000} C_DIS
LIN {X 96.718,Y 59.257,Z 64.500,A 180.000,B 0.000,C 180.000} C_DIS
LIN {X 96.883,Y 59.176,Z 64.500,A 180.000,B 0.000,C 180.000} C_DIS
LIN {X 96.897,Y 59.169,Z 64.500,A 180.000,B 0.000,C 180.000} C_DIS
LIN {X 97.075,Y 59.061,Z 64.500,A 180.000,B 0.000,C 180.000} C_DIS
LIN {X 97.167,Y 58.997,Z 64.500,A 180.000,B 0.000,C 180.000} C_DIS
LIN {X 97.210,Y 58.965,Z 64.500,A 180.000,B 0.000,C 180.000} C_DIS
LIN {X 97.232,Y 58.948,Z 64.500,A 180.000,B 0.000,C 180.000} C_DIS
LIN {X 97.243,Y 58.939,Z 64.500,A 180.000,B 0.000,C 180.000} C_DIS
LIN {X 97.250,Y 58.934,Z 64.500,A 180.000,B 0.000,C 180.000} C_DIS
LIN {X 97.251,Y 58.933,Z 64.500,A 180.000,B 0.000,C 180.000} C_DIS
LIN {X 97.254,Y 58.932,Z 64.500,A 180.000,B 0.000,C 180.000} C_DIS
LIN {X 97.790,Y 58.693,Z 64.500,A 180.000,B 0.000,C 180.000} C_DIS
LIN {X 97.906,Y 58.640,Z 64.500,A 180.000,B 0.000,C 180.000} C_DIS
LIN {X 97.969,Y 58.608,Z 64.500,A 180.000,B 0.000,C 180.000} C_DIS
LIN {X 98.505,Y 58.327,Z 64.500,A 180.000,B 0.000,C 180.000} C_DIS
LIN {X 98.588,Y 58.282,Z 64.500,A 180.000,B 0.000,C 180.000} C_DIS
LIN {X 98.684,Y 58.225,Z 64.500,A 180.000,B 0.000,C 180.000} C_DIS
LIN {X 99.179,Y 57.925,Z 64.500,A 180.000,B 0.000,C 180.000} C_DIS
LIN {X 99.221,Y 57.899,Z 64.500,A 180.000,B 0.000,C 180.000} C_DIS
LIN {X 99.399,Y 57.778,Z 64.500,A 180.000,B 0.000,C 180.000} C_DIS
LIN {X 99.757,Y 57.529,Z 64.500,A 180.000,B 0.000,C 180.000} C_DIS
LIN {X 99.936,Y 57.400,Z 64.500,A 180.000,B 0.000,C 180.000} C_DIS
LIN {X 99.951,Y 57.388,Z 64.500,A 180.000,B 0.000,C 180.000} C_DIS
LIN {X 100.401,Y 57.031,Z 64.500,A 180.000,B 0.000,C 180.000} C_DIS
LIN {X 100.472,Y 56.974,Z 64.500,A 180.000,B 0.000,C 180.000} C_DIS
LIN {X 100.611,Y 56.852,Z 64.500,A 180.000,B 0.000,C 180.000} C_DIS
LIN {X 101.008,Y 56.494,Z 64.500,A 180.000,B 0.000,C 180.000} C_DIS
LIN {X 101.187,Y 56.320,Z 64.500,A 180.000,B 0.000,C 180.000} C_DIS
LIN {X 101.545,Y 55.954,Z 64.500,A 180.000,B 0.000,C 180.000} C_DIS
LIN {X 101.704,Y 55.779,Z 64.500,A 180.000,B 0.000,C 180.000} C_DIS
LIN {X 102.081,Y 55.342,Z 64.500,A 180.000,B 0.000,C 180.000} C_DIS
LIN {X 102.162,Y 55.243,Z 64.500,A 180.000,B 0.000,C 180.000} C_DIS
LIN {X 102.260,Y 55.114,Z 64.500,A 180.000,B 0.000,C 180.000} C_DIS
LIN {X 102.438,Y 54.878,Z 64.500,A 180.000,B 0.000,C 180.000} C_DIS
LIN {X 102.568,Y 54.707,Z 64.500,A 180.000,B 0.000,C 180.000} C_DIS
LIN {X 102.617,Y 54.638,Z 64.500,A 180.000,B 0.000,C 180.000} C_DIS
LIN {X 102.691,Y 54.528,Z 64.500,A 180.000,B 0.000,C 180.000} C_DIS
LIN {X 102.975,Y 54.100,Z 64.500,A 180.000,B 0.000,C 180.000} C_DIS
LIN {X 103.044,Y 53.992,Z 64.500,A 180.000,B 0.000,C 180.000} C_DIS
LIN {X 103.147,Y 53.813,Z 64.500,A 180.000,B 0.000,C 180.000} C_DIS
LIN {X 103.353,Y 53.455,Z 64.500,A 180.000,B 0.000,C 180.000} C_DIS
LIN {X 103.451,Y 53.277,Z 64.500,A 180.000,B 0.000,C 180.000} C_DIS
LIN {X 103.717,Y 52.740,Z 64.500,A 180.000,B 0.000,C 180.000} C_DIS
LIN {X 103.799,Y 52.562,Z 64.500,A 180.000,B 0.000,C 180.000} C_DIS
LIN {X 104.024,Y 52.025,Z 64.500,A 180.000,B 0.000,C 180.000} C_DIS
LIN {X 104.047,Y 51.968,Z 64.500,A 180.000,B 0.000,C 180.000} C_DIS
LIN {X 104.093,Y 51.847,Z 64.500,A 180.000,B 0.000,C 180.000} C_DIS
LIN {X 104.279,Y 51.310,Z 64.500,A 180.000,B 0.000,C 180.000} C_DIS
LIN {X 104.337,Y 51.131,Z 64.500,A 180.000,B 0.000,C 180.000} C_DIS
LIN {X 104.387,Y 50.953,Z 64.500,A 180.000,B 0.000,C 180.000} C_DIS
LIN {X 104.486,Y 50.595,Z 64.500,A 180.000,B 0.000,C 180.000} C_DIS
LIN {X 104.534,Y 50.416,Z 64.500,A 180.000,B 0.000,C 180.000} C_DIS
LIN {X 104.572,Y 50.238,Z 64.500,A 180.000,B 0.000,C 180.000} C_DIS
LIN {X 104.648,Y 49.880,Z 64.500,A 180.000,B 0.000,C 180.000} C_DIS
LIN {X 104.685,Y 49.701,Z 64.500,A 180.000,B 0.000,C 180.000} C_DIS
LIN {X 104.713,Y 49.523,Z 64.500,A 180.000,B 0.000,C 180.000} C_DIS
LIN {X 104.792,Y 48.986,Z 64.500,A 180.000,B 0.000,C 180.000} C_DIS
LIN {X 104.811,Y 48.807,Z 64.500,A 180.000,B 0.000,C 180.000} C_DIS
LIN {X 104.856,Y 48.271,Z 64.500,A 180.000,B 0.000,C 180.000} C_DIS
LIN {X 104.868,Y 48.092,Z 64.500,A 180.000,B 0.000,C 180.000} C_DIS
LIN {X 104.871,Y 47.914,Z 64.500,A 180.000,B 0.000,C 180.000} C_DIS
LIN {X 104.879,Y 47.556,Z 64.500,A 180.000,B 0.000,C 180.000} C_DIS
LIN {X 104.881,Y 47.377,Z 64.500,A 180.000,B 0.000,C 180.000} C_DIS
LIN {X 104.876,Y 47.198,Z 64.500,A 180.000,B 0.000,C 180.000} C_DIS
LIN {X 104.853,Y 46.662,Z 64.500,A 180.000,B 0.000,C 180.000} C_DIS
LIN {X 104.839,Y 46.483,Z 64.500,A 180.000,B 0.000,C 180.000} C_DIS
LIN {X 104.782,Y 45.947,Z 64.500,A 180.000,B 0.000,C 180.000} C_DIS
LIN {X 104.762,Y 45.784,Z 64.500,A 180.000,B 0.000,C 180.000} C_DIS
LIN {X 104.760,Y 45.768,Z 64.500,A 180.000,B 0.000,C 180.000} C_DIS
LIN {X 104.730,Y 45.590,Z 64.500,A 180.000,B 0.000,C 180.000} C_DIS
LIN {X 104.669,Y 45.232,Z 64.500,A 180.000,B 0.000,C 180.000} C_DIS
LIN {X 104.638,Y 45.053,Z 64.500,A 180.000,B 0.000,C 180.000} C_DIS
LIN {X 104.597,Y 44.874,Z 64.500,A 180.000,B 0.000,C 180.000} C_DIS
LIN {X 104.513,Y 44.517,Z 64.500,A 180.000,B 0.000,C 180.000} C_DIS
LIN {X 104.471,Y 44.338,Z 64.500,A 180.000,B 0.000,C 180.000} C_DIS
LIN {X 104.421,Y 44.159,Z 64.500,A 180.000,B 0.000,C 180.000} C_DIS
LIN {X 104.258,Y 43.623,Z 64.500,A 180.000,B 0.000,C 180.000} C_DIS
LIN {X 104.226,Y 43.524,Z 64.500,A 180.000,B 0.000,C 180.000} C_DIS
LIN {X 104.197,Y 43.444,Z 64.500,A 180.000,B 0.000,C 180.000} C_DIS
LIN {X 103.997,Y 42.908,Z 64.500,A 180.000,B 0.000,C 180.000} C_DIS
LIN {X 103.925,Y 42.729,Z 64.500,A 180.000,B 0.000,C 180.000} C_DIS
LIN {X 103.685,Y 42.193,Z 64.500,A 180.000,B 0.000,C 180.000} C_DIS
LIN {X 103.599,Y 42.014,Z 64.500,A 180.000,B 0.000,C 180.000} C_DIS
LIN {X 103.332,Y 41.505,Z 64.500,A 180.000,B 0.000,C 180.000} C_DIS
LIN {X 103.318,Y 41.478,Z 64.500,A 180.000,B 0.000,C 180.000} C_DIS
LIN {X 103.215,Y 41.299,Z 64.500,A 180.000,B 0.000,C 180.000} C_DIS
LIN {X 102.975,Y 40.903,Z 64.500,A 180.000,B 0.000,C 180.000} C_DIS
LIN {X 102.889,Y 40.763,Z 64.500,A 180.000,B 0.000,C 180.000} C_DIS
LIN {X 102.796,Y 40.626,Z 64.500,A 180.000,B 0.000,C 180.000} C_DIS
LIN {X 102.518,Y 40.226,Z 64.500,A 180.000,B 0.000,C 180.000} C_DIS
LIN {X 102.438,Y 40.115,Z 64.500,A 180.000,B 0.000,C 180.000} C_DIS
LIN {X 102.387,Y 40.048,Z 64.500,A 180.000,B 0.000,C 180.000} C_DIS
LIN {X 102.081,Y 39.662,Z 64.500,A 180.000,B 0.000,C 180.000} C_DIS
LIN {X 101.960,Y 39.511,Z 64.500,A 180.000,B 0.000,C 180.000} C_DIS
LIN {X 101.902,Y 39.444,Z 64.500,A 180.000,B 0.000,C 180.000} C_DIS
LIN {X 101.545,Y 39.048,Z 64.500,A 180.000,B 0.000,C 180.000} C_DIS
LIN {X 101.479,Y 38.975,Z 64.500,A 180.000,B 0.000,C 180.000} C_DIS
LIN {X 101.366,Y 38.858,Z 64.500,A 180.000,B 0.000,C 180.000} C_DIS
LIN {X 100.937,Y 38.439,Z 64.500,A 180.000,B 0.000,C 180.000} C_DIS
LIN {X 100.829,Y 38.339,Z 64.500,A 180.000,B 0.000,C 180.000} C_DIS
LIN {X 100.738,Y 38.260,Z 64.500,A 180.000,B 0.000,C 180.000} C_DIS
LIN {X 100.472,Y 38.031,Z 64.500,A 180.000,B 0.000,C 180.000} C_DIS
LIN {X 100.323,Y 37.902,Z 64.500,A 180.000,B 0.000,C 180.000} C_DIS
LIN {X 100.293,Y 37.878,Z 64.500,A 180.000,B 0.000,C 180.000} C_DIS
LIN {X 100.114,Y 37.741,Z 64.500,A 180.000,B 0.000,C 180.000} C_DIS
LIN {X 99.757,Y 37.470,Z 64.500,A 180.000,B 0.000,C 180.000} C_DIS
LIN {X 99.614,Y 37.366,Z 64.500,A 180.000,B 0.000,C 180.000} C_DIS
LIN {X 99.578,Y 37.342,Z 64.500,A 180.000,B 0.000,C 180.000} C_DIS
LIN {X 99.221,Y 37.105,Z 64.500,A 180.000,B 0.000,C 180.000} C_DIS
LIN {X 99.075,Y 37.009,Z 64.500,A 180.000,B 0.000,C 180.000} C_DIS
LIN {X 99.042,Y 36.987,Z 64.500,A 180.000,B 0.000,C 180.000} C_DIS
LIN {X 98.863,Y 36.882,Z 64.500,A 180.000,B 0.000,C 180.000} C_DIS
LIN {X 98.463,Y 36.651,Z 64.500,A 180.000,B 0.000,C 180.000} C_DIS
LIN {X 98.327,Y 36.575,Z 64.500,A 180.000,B 0.000,C 180.000} C_DIS
LIN {X 98.148,Y 36.485,Z 64.500,A 180.000,B 0.000,C 180.000} C_DIS
LIN {X 97.761,Y 36.294,Z 64.500,A 180.000,B 0.000,C 180.000} C_DIS
LIN {X 97.612,Y 36.223,Z 64.500,A 180.000,B 0.000,C 180.000} C_DIS
LIN {X 97.433,Y 36.147,Z 64.500,A 180.000,B 0.000,C 180.000} C_DIS
LIN {X 97.075,Y 35.997,Z 64.500,A 180.000,B 0.000,C 180.000} C_DIS
LIN {X 96.926,Y 35.936,Z 64.500,A 180.000,B 0.000,C 180.000} C_DIS
LIN {X 96.897,Y 35.925,Z 64.500,A 180.000,B 0.000,C 180.000} C_DIS
LIN {X 96.718,Y 35.862,Z 64.500,A 180.000,B 0.000,C 180.000} C_DIS
LIN {X 96.360,Y 35.738,Z 64.500,A 180.000,B 0.000,C 180.000} C_DIS
LIN {X 96.181,Y 35.678,Z 64.500,A 180.000,B 0.000,C 180.000} C_DIS
LIN {X 96.003,Y 35.627,Z 64.500,A 180.000,B 0.000,C 180.000} C_DIS
LIN {X 95.645,Y 35.528,Z 64.500,A 180.000,B 0.000,C 180.000} C_DIS
LIN {X 95.466,Y 35.479,Z 64.500,A 180.000,B 0.000,C 180.000} C_DIS
LIN {X 95.288,Y 35.439,Z 64.500,A 180.000,B 0.000,C 180.000} C_DIS
LIN {X 94.930,Y 35.363,Z 64.500,A 180.000,B 0.000,C 180.000} C_DIS
LIN {X 94.751,Y 35.325,Z 64.500,A 180.000,B 0.000,C 180.000} C_DIS
LIN {X 94.573,Y 35.294,Z 64.500,A 180.000,B 0.000,C 180.000} C_DIS
LIN {X 94.036,Y 35.216,Z 64.500,A 180.000,B 0.000,C 180.000} C_DIS
LIN {X 93.857,Y 35.193,Z 64.500,A 180.000,B 0.000,C 180.000} C_DIS
LIN {X 93.679,Y 35.178,Z 64.500,A 180.000,B 0.000,C 180.000} C_DIS
LIN {X 93.321,Y 35.148,Z 64.500,A 180.000,B 0.000,C 180.000} C_DIS
LIN {X 93.142,Y 35.135,Z 64.500,A 180.000,B 0.000,C 180.000} C_DIS
LIN {X 92.964,Y 35.130,Z 64.500,A 180.000,B 0.000,C 180.000} C_DIS
LIN {X 92.606,Y 35.122,Z 64.500,A 180.000,B 0.000,C 180.000} C_DIS
LIN {X 92.427,Y 35.119,Z 64.500,A 180.000,B 0.000,C 180.000} C_DIS
LIN {X 92.249,Y 35.122,Z 64.500,A 180.000,B 0.000,C 180.000} C_DIS
LIN {X 91.712,Y 35.145,Z 64.500,A 180.000,B 0.000,C 180.000} C_DIS
LIN {X 91.533,Y 35.156,Z 64.500,A 180.000,B 0.000,C 180.000} C_DIS
LIN {X 91.355,Y 35.175,Z 64.500,A 180.000,B 0.000,C 180.000} C_DIS
LIN {X 90.920,Y 35.221,Z 64.500,A 180.000,B 0.000,C 180.000} C_DIS
LIN {X 90.818,Y 35.233,Z 64.500,A 180.000,B 0.000,C 180.000} C_DIS
LIN {X 90.640,Y 35.262,Z 64.500,A 180.000,B 0.000,C 180.000} C_DIS
LIN {X 90.282,Y 35.322,Z 64.500,A 180.000,B 0.000,C 180.000} C_DIS
LIN {X 90.103,Y 35.353,Z 64.500,A 180.000,B 0.000,C 180.000} C_DIS
LIN {X 89.925,Y 35.391,Z 64.500,A 180.000,B 0.000,C 180.000} C_DIS
LIN {X 89.366,Y 35.522,Z 64.500,A 180.000,B 0.000,C 180.000} C_DIS
LIN {X 89.355,Y 35.525,Z 64.500,A 180.000,B 0.000,C 180.000} C_DIS
LIN {X 89.353,Y 35.525,Z 64.500,A 180.000,B 0.000,C 180.000} C_DIS
LIN {X 89.344,Y 35.525,Z 64.500,A 180.000,B 0.000,C 180.000} C_DIS
LIN {X 89.299,Y 35.525,Z 64.500,A 180.000,B 0.000,C 180.000} C_DIS
LIN {X 89.209,Y 35.526,Z 64.500,A 180.000,B 0.000,C 180.000} C_DIS
LIN {X 89.031,Y 35.540,Z 64.500,A 180.000,B 0.000,C 180.000} C_DIS
LIN {X 88.852,Y 35.566,Z 64.500,A 180.000,B 0.000,C 180.000} C_DIS
LIN {X 88.788,Y 35.578,Z 64.500,A 180.000,B 0.000,C 180.000} C_DIS
LIN {X 88.673,Y 35.605,Z 64.500,A 180.000,B 0.000,C 180.000} C_DIS
LIN {X 88.494,Y 35.659,Z 64.500,A 180.000,B 0.000,C 180.000} C_DIS
LIN {X 55.704,Y 46.721,Z 64.500,A 180.000,B 0.000,C 180.000} C_DIS
LIN {X 45.590,Y 50.133,Z 64.500,A 180.000,B 0.000,C 180.000} C_DIS
LIN {X 45.411,Y 50.194,Z 64.500,A 180.000,B 0.000,C 180.000} C_DIS
LIN {X 45.296,Y 50.238,Z 64.500,A 180.000,B 0.000,C 180.000} C_DIS
LIN {X 45.232,Y 50.265,Z 64.500,A 180.000,B 0.000,C 180.000} C_DIS
LIN {X 45.053,Y 50.353,Z 64.500,A 180.000,B 0.000,C 180.000} C_DIS
LIN {X 44.944,Y 50.416,Z 64.500,A 180.000,B 0.000,C 180.000} C_DIS
LIN {X 44.874,Y 50.461,Z 64.500,A 180.000,B 0.000,C 180.000} C_DIS
LIN {X 44.785,Y 50.522,Z 64.500,A 180.000,B 0.000,C 180.000} C_DIS
LIN {X 44.696,Y 50.590,Z 64.500,A 180.000,B 0.000,C 180.000} C_DIS
LIN {X 44.689,Y 50.595,Z 64.500,A 180.000,B 0.000,C 180.000} C_DIS
LIN {X 44.603,Y 50.667,Z 64.500,A 180.000,B 0.000,C 180.000} C_DIS
LIN {X 44.517,Y 50.746,Z 64.500,A 180.000,B 0.000,C 180.000} C_DIS
LIN {X 44.488,Y 50.774,Z 64.500,A 180.000,B 0.000,C 180.000} C_DIS
LIN {X 44.410,Y 50.855,Z 64.500,A 180.000,B 0.000,C 180.000} C_DIS
LIN {X 44.338,Y 50.936,Z 64.500,A 180.000,B 0.000,C 180.000} C_DIS
LIN {X 44.325,Y 50.953,Z 64.500,A 180.000,B 0.000,C 180.000} C_DIS
LIN {X 44.254,Y 51.042,Z 64.500,A 180.000,B 0.000,C 180.000} C_DIS
LIN {X 44.189,Y 51.131,Z 64.500,A 180.000,B 0.000,C 180.000} C_DIS
LIN {X 44.159,Y 51.176,Z 64.500,A 180.000,B 0.000,C 180.000} C_DIS
LIN {X 44.077,Y 51.310,Z 64.500,A 180.000,B 0.000,C 180.000} C_DIS
LIN {X 43.984,Y 51.489,Z 64.500,A 180.000,B 0.000,C 180.000} C_DIS
LIN {X 43.981,Y 51.497,Z 64.500,A 180.000,B 0.000,C 180.000} C_DIS
LIN {X 43.909,Y 51.668,Z 64.500,A 180.000,B 0.000,C 180.000} C_DIS
LIN {X 43.849,Y 51.847,Z 64.500,A 180.000,B 0.000,C 180.000} C_DIS
LIN {X 43.804,Y 52.025,Z 64.500,A 180.000,B 0.000,C 180.000} C_DIS
LIN {X 43.802,Y 52.035,Z 64.500,A 180.000,B 0.000,C 180.000} C_DIS
LIN {X 43.772,Y 52.204,Z 64.500,A 180.000,B 0.000,C 180.000} C_DIS
LIN {X 43.754,Y 52.383,Z 64.500,A 180.000,B 0.000,C 180.000} C_DIS
LIN {X 43.748,Y 52.562,Z 64.500,A 180.000,B 0.000,C 180.000} C_DIS
LIN {X 43.756,Y 52.740,Z 64.500,A 180.000,B 0.000,C 180.000} C_DIS
LIN {X 43.776,Y 52.919,Z 64.500,A 180.000,B 0.000,C 180.000} C_DIS
LIN {X 43.802,Y 53.064,Z 64.500,A 180.000,B 0.000,C 180.000} C_DIS
LIN {X 43.809,Y 53.098,Z 64.500,A 180.000,B 0.000,C 180.000} C_DIS
LIN {X 43.856,Y 53.277,Z 64.500,A 180.000,B 0.000,C 180.000} C_DIS
LIN {X 43.916,Y 53.455,Z 64.500,A 180.000,B 0.000,C 180.000} C_DIS
LIN {X 50.248,Y 72.226,Z 64.500,A 180.000,B 0.000,C 180.000} C_DIS
LIN {X 50.311,Y 72.405,Z 64.500,A 180.000,B 0.000,C 180.000} C_DIS
LIN {X 50.388,Y 72.584,Z 64.500,A 180.000,B 0.000,C 180.000} C_DIS
LIN {X 50.416,Y 72.640,Z 64.500,A 180.000,B 0.000,C 180.000} C_DIS
LIN {X 50.484,Y 72.763,Z 64.500,A 180.000,B 0.000,C 180.000} C_DIS
LIN {X 50.595,Y 72.936,Z 64.500,A 180.000,B 0.000,C 180.000} C_DIS
LIN {X 50.599,Y 72.941,Z 64.500,A 180.000,B 0.000,C 180.000} C_DIS
LIN {X 50.665,Y 73.031,Z 64.500,A 180.000,B 0.000,C 180.000} C_DIS
LIN {X 50.737,Y 73.120,Z 64.500,A 180.000,B 0.000,C 180.000} C_DIS
LIN {X 50.774,Y 73.162,Z 64.500,A 180.000,B 0.000,C 180.000} C_DIS
LIN {X 50.905,Y 73.299,Z 64.500,A 180.000,B 0.000,C 180.000} C_DIS
LIN {X 50.953,Y 73.343,Z 64.500,A 180.000,B 0.000,C 180.000} C_DIS
LIN {X 51.112,Y 73.478,Z 64.500,A 180.000,B 0.000,C 180.000} C_DIS
LIN {X 51.131,Y 73.493,Z 64.500,A 180.000,B 0.000,C 180.000} C_DIS
LIN {X 51.310,Y 73.616,Z 64.500,A 180.000,B 0.000,C 180.000} C_DIS
LIN {X 51.376,Y 73.656,Z 64.500,A 180.000,B 0.000,C 180.000} C_DIS
LIN {X 51.489,Y 73.719,Z 64.500,A 180.000,B 0.000,C 180.000} C_DIS
LIN {X 51.668,Y 73.803,Z 64.500,A 180.000,B 0.000,C 180.000} C_DIS
LIN {X 51.749,Y 73.835,Z 64.500,A 180.000,B 0.000,C 180.000} C_DIS
LIN {X 51.847,Y 73.870,Z 64.500,A 180.000,B 0.000,C 180.000} C_DIS
LIN {X 51.880,Y 73.880,Z 64.500,A 180.000,B 0.000,C 180.000} C_DIS
; Link Move Starts
LIN {X 52.031,Y 73.924,Z 64.500,A 180.000,B 0.000,C 180.000} C_DIS
LIN {X 52.185,Y 73.958,Z 64.500,A 180.000,B 0.000,C 180.000} C_DIS
LIN {X 52.341,Y 73.982,Z 64.499,A 180.000,B 0.000,C 180.000} C_DIS
LIN {X 52.497,Y 73.996,Z 64.499,A 180.000,B 0.000,C 180.000} C_DIS
LIN {X 52.655,Y 74.000,Z 64.498,A 180.000,B 0.000,C 180.000} C_DIS
LIN {X 52.812,Y 73.994,Z 64.498,A 180.000,B 0.000,C 180.000} C_DIS
LIN {X 52.969,Y 73.978,Z 64.497,A 180.000,B 0.000,C 180.000} C_DIS
LIN {X 53.124,Y 73.953,Z 64.496,A 180.000,B 0.000,C 180.000} C_DIS
LIN {X 53.278,Y 73.918,Z 64.495,A 180.000,B 0.000,C 180.000} C_DIS
LIN {X 53.429,Y 73.873,Z 64.494,A 180.000,B 0.000,C 180.000} C_DIS
LIN {X 53.727,Y 73.772,Z 64.491,A 180.000,B 0.000,C 180.000} C_DIS
LIN {X 54.026,Y 73.671,Z 64.488,A 180.000,B 0.000,C 180.000} C_DIS
LIN {X 54.324,Y 73.571,Z 64.485,A 180.000,B 0.000,C 180.000} C_DIS
LIN {X 54.623,Y 73.470,Z 64.481,A 180.000,B 0.000,C 180.000} C_DIS
LIN {X 54.921,Y 73.369,Z 64.477,A 180.000,B 0.000,C 180.000} C_DIS
LIN {X 55.220,Y 73.269,Z 64.472,A 180.000,B 0.000,C 180.000} C_DIS
LIN {X 55.369,Y 73.218,Z 64.469,A 180.000,B 0.000,C 180.000} C_DIS
LIN {X 55.518,Y 73.168,Z 64.467,A 180.000,B 0.000,C 180.000} C_DIS
LIN {X 55.667,Y 73.118,Z 64.464,A 180.000,B 0.000,C 180.000} C_DIS
LIN {X 55.817,Y 73.067,Z 64.461,A 180.000,B 0.000,C 180.000} C_DIS
LIN {X 55.966,Y 73.017,Z 64.459,A 180.000,B 0.000,C 180.000} C_DIS
LIN {X 56.115,Y 72.967,Z 64.456,A 180.000,B 0.000,C 180.000} C_DIS
LIN {X 56.264,Y 72.916,Z 64.452,A 180.000,B 0.000,C 180.000} C_DIS
LIN {X 56.414,Y 72.866,Z 64.449,A 180.000,B 0.000,C 180.000} C_DIS
LIN {X 56.563,Y 72.815,Z 64.446,A 180.000,B 0.000,C 180.000} C_DIS
LIN {X 56.712,Y 72.765,Z 64.443,A 180.000,B 0.000,C 180.000} C_DIS
LIN {X 56.861,Y 72.715,Z 64.439,A 180.000,B 0.000,C 180.000} C_DIS
LIN {X 57.011,Y 72.664,Z 64.436,A 180.000,B 0.000,C 180.000} C_DIS
LIN {X 57.160,Y 72.614,Z 64.432,A 180.000,B 0.000,C 180.000} C_DIS
LIN {X 57.309,Y 72.564,Z 64.428,A 180.000,B 0.000,C 180.000} C_DIS
LIN {X 57.458,Y 72.513,Z 64.425,A 180.000,B 0.000,C 180.000} C_DIS
LIN {X 57.608,Y 72.463,Z 64.421,A 180.000,B 0.000,C 180.000} C_DIS
LIN {X 57.757,Y 72.413,Z 64.417,A 180.000,B 0.000,C 180.000} C_DIS
LIN {X 57.906,Y 72.362,Z 64.413,A 180.000,B 0.000,C 180.000} C_DIS
LIN {X 58.055,Y 72.312,Z 64.409,A 180.000,B 0.000,C 180.000} C_DIS
LIN {X 58.204,Y 72.262,Z 64.405,A 180.000,B 0.000,C 180.000} C_DIS
LIN {X 58.354,Y 72.211,Z 64.400,A 180.000,B 0.000,C 180.000} C_DIS
LIN {X 58.503,Y 72.161,Z 64.396,A 180.000,B 0.000,C 180.000} C_DIS
LIN {X 58.652,Y 72.111,Z 64.392,A 180.000,B 0.000,C 180.000} C_DIS
LIN {X 58.801,Y 72.060,Z 64.387,A 180.000,B 0.000,C 180.000} C_DIS
LIN {X 58.951,Y 72.010,Z 64.383,A 180.000,B 0.000,C 180.000} C_DIS
LIN {X 59.100,Y 71.960,Z 64.378,A 180.000,B 0.000,C 180.000} C_DIS
LIN {X 59.249,Y 71.909,Z 64.373,A 180.000,B 0.000,C 180.000} C_DIS
LIN {X 59.398,Y 71.859,Z 64.369,A 180.000,B 0.000,C 180.000} C_DIS
LIN {X 59.548,Y 71.809,Z 64.364,A 180.000,B 0.000,C 180.000} C_DIS
LIN {X 59.697,Y 71.758,Z 64.359,A 180.000,B 0.000,C 180.000} C_DIS
LIN {X 59.846,Y 71.708,Z 64.354,A 180.000,B 0.000,C 180.000} C_DIS
LIN {X 59.921,Y 71.683,Z 64.351,A 180.000,B 0.000,C 180.000} C_DIS
LIN {X 59.995,Y 71.658,Z 64.349,A 180.000,B 0.000,C 180.000} C_DIS
LIN {X 60.070,Y 71.632,Z 64.346,A 180.000,B 0.000,C 180.000} C_DIS
LIN {X 60.145,Y 71.607,Z 64.344,A 180.000,B 0.000,C 180.000} C_DIS
LIN {X 60.219,Y 71.582,Z 64.341,A 180.000,B 0.000,C 180.000} C_DIS
LIN {X 60.294,Y 71.557,Z 64.339,A 180.000,B 0.000,C 180.000} C_DIS
LIN {X 60.368,Y 71.532,Z 64.336,A 180.000,B 0.000,C 180.000} C_DIS
LIN {X 60.518,Y 71.481,Z 64.331,A 180.000,B 0.000,C 180.000} C_DIS
LIN {X 60.667,Y 71.431,Z 64.325,A 180.000,B 0.000,C 180.000} C_DIS
LIN {X 60.816,Y 71.381,Z 64.320,A 180.000,B 0.000,C 180.000} C_DIS
LIN {X 60.965,Y 71.330,Z 64.315,A 180.000,B 0.000,C 180.000} C_DIS
LIN {X 61.115,Y 71.280,Z 64.309,A 180.000,B 0.000,C 180.000} C_DIS
LIN {X 61.189,Y 71.255,Z 64.307,A 180.000,B 0.000,C 180.000} C_DIS
LIN {X 61.338,Y 71.204,Z 64.301,A 180.000,B 0.000,C 180.000} C_DIS
LIN {X 61.562,Y 71.129,Z 64.293,A 180.000,B 0.000,C 180.000} C_DIS
LIN {X 61.712,Y 71.079,Z 64.287,A 180.000,B 0.000,C 180.000} C_DIS
LIN {X 61.786,Y 71.053,Z 64.285,A 180.000,B 0.000,C 180.000} C_DIS
LIN {X 61.935,Y 71.003,Z 64.279,A 180.000,B 0.000,C 180.000} C_DIS
LIN {X 62.159,Y 70.928,Z 64.271,A 180.000,B 0.000,C 180.000} C_DIS
LIN {X 62.308,Y 70.877,Z 64.265,A 180.000,B 0.000,C 180.000} C_DIS
LIN {X 62.383,Y 70.852,Z 64.263,A 180.000,B 0.000,C 180.000} C_DIS
LIN {X 62.532,Y 70.802,Z 64.257,A 180.000,B 0.000,C 180.000} C_DIS
LIN {X 62.756,Y 70.726,Z 64.249,A 180.000,B 0.000,C 180.000} C_DIS
LIN {X 62.905,Y 70.676,Z 64.243,A 180.000,B 0.000,C 180.000} C_DIS
LIN {X 62.980,Y 70.651,Z 64.241,A 180.000,B 0.000,C 180.000} C_DIS
LIN {X 63.129,Y 70.600,Z 64.235,A 180.000,B 0.000,C 180.000} C_DIS
LIN {X 63.353,Y 70.525,Z 64.227,A 180.000,B 0.000,C 180.000} C_DIS
LIN {X 63.502,Y 70.474,Z 64.221,A 180.000,B 0.000,C 180.000} C_DIS
LIN {X 63.577,Y 70.449,Z 64.219,A 180.000,B 0.000,C 180.000} C_DIS
LIN {X 63.726,Y 70.399,Z 64.213,A 180.000,B 0.000,C 180.000} C_DIS
LIN {X 64.174,Y 70.248,Z 64.197,A 180.000,B 0.000,C 180.000} C_DIS
LIN {X 64.323,Y 70.198,Z 64.191,A 180.000,B 0.000,C 180.000} C_DIS
LIN {X 64.771,Y 70.047,Z 64.175,A 180.000,B 0.000,C 180.000} C_DIS
LIN {X 64.920,Y 69.996,Z 64.169,A 180.000,B 0.000,C 180.000} C_DIS
LIN {X 65.442,Y 69.820,Z 64.150,A 180.000,B 0.000,C 180.000} C_DIS
LIN {X 65.890,Y 69.669,Z 64.133,A 180.000,B 0.000,C 180.000} C_DIS
LIN {X 66.039,Y 69.619,Z 64.128,A 180.000,B 0.000,C 180.000} C_DIS
LIN {X 66.487,Y 69.468,Z 64.111,A 180.000,B 0.000,C 180.000} C_DIS
LIN {X 66.636,Y 69.417,Z 64.106,A 180.000,B 0.000,C 180.000} C_DIS
LIN {X 67.382,Y 69.165,Z 64.078,A 180.000,B 0.000,C 180.000} C_DIS
LIN {X 67.756,Y 69.040,Z 64.065,A 180.000,B 0.000,C 180.000} C_DIS
LIN {X 68.203,Y 68.889,Z 64.048,A 180.000,B 0.000,C 180.000} C_DIS
LIN {X 69.919,Y 68.310,Z 63.985,A 180.000,B 0.000,C 180.000} C_DIS
LIN {X 72.755,Y 67.353,Z 63.880,A 180.000,B 0.000,C 180.000} C_DIS
LIN {X 72.904,Y 67.303,Z 63.875,A 180.000,B 0.000,C 180.000} C_DIS
LIN {X 73.352,Y 67.152,Z 63.858,A 180.000,B 0.000,C 180.000} C_DIS
LIN {X 73.501,Y 67.101,Z 63.853,A 180.000,B 0.000,C 180.000} C_DIS
LIN {X 73.949,Y 66.950,Z 63.836,A 180.000,B 0.000,C 180.000} C_DIS
LIN {X 74.023,Y 66.925,Z 63.834,A 180.000,B 0.000,C 180.000} C_DIS
LIN {X 74.173,Y 66.875,Z 63.828,A 180.000,B 0.000,C 180.000} C_DIS
LIN {X 74.620,Y 66.724,Z 63.812,A 180.000,B 0.000,C 180.000} C_DIS
LIN {X 74.770,Y 66.673,Z 63.806,A 180.000,B 0.000,C 180.000} C_DIS
LIN {X 75.217,Y 66.522,Z 63.790,A 180.000,B 0.000,C 180.000} C_DIS
LIN {X 75.367,Y 66.472,Z 63.784,A 180.000,B 0.000,C 180.000} C_DIS
LIN {X 75.590,Y 66.397,Z 63.776,A 180.000,B 0.000,C 180.000} C_DIS
LIN {X 75.740,Y 66.346,Z 63.770,A 180.000,B 0.000,C 180.000} C_DIS
LIN {X 75.814,Y 66.321,Z 63.768,A 180.000,B 0.000,C 180.000} C_DIS
LIN {X 75.964,Y 66.271,Z 63.762,A 180.000,B 0.000,C 180.000} C_DIS
LIN {X 76.187,Y 66.195,Z 63.754,A 180.000,B 0.000,C 180.000} C_DIS
LIN {X 76.337,Y 66.145,Z 63.748,A 180.000,B 0.000,C 180.000} C_DIS
LIN {X 76.411,Y 66.120,Z 63.746,A 180.000,B 0.000,C 180.000} C_DIS
LIN {X 76.561,Y 66.069,Z 63.740,A 180.000,B 0.000,C 180.000} C_DIS
LIN {X 76.784,Y 65.994,Z 63.732,A 180.000,B 0.000,C 180.000} C_DIS
LIN {X 76.934,Y 65.943,Z 63.726,A 180.000,B 0.000,C 180.000} C_DIS
LIN {X 77.008,Y 65.918,Z 63.724,A 180.000,B 0.000,C 180.000} C_DIS
LIN {X 77.157,Y 65.868,Z 63.718,A 180.000,B 0.000,C 180.000} C_DIS
LIN {X 77.381,Y 65.792,Z 63.710,A 180.000,B 0.000,C 180.000} C_DIS
LIN {X 77.531,Y 65.742,Z 63.704,A 180.000,B 0.000,C 180.000} C_DIS
LIN {X 77.605,Y 65.717,Z 63.702,A 180.000,B 0.000,C 180.000} C_DIS
LIN {X 77.754,Y 65.667,Z 63.696,A 180.000,B 0.000,C 180.000} C_DIS
LIN {X 77.904,Y 65.616,Z 63.691,A 180.000,B 0.000,C 180.000} C_DIS
LIN {X 78.053,Y 65.566,Z 63.685,A 180.000,B 0.000,C 180.000} C_DIS
LIN {X 78.202,Y 65.516,Z 63.680,A 180.000,B 0.000,C 180.000} C_DIS
LIN {X 78.351,Y 65.465,Z 63.674,A 180.000,B 0.000,C 180.000} C_DIS
LIN {X 78.501,Y 65.415,Z 63.669,A 180.000,B 0.000,C 180.000} C_DIS
LIN {X 78.650,Y 65.364,Z 63.664,A 180.000,B 0.000,C 180.000} C_DIS
LIN {X 78.724,Y 65.339,Z 63.661,A 180.000,B 0.000,C 180.000} C_DIS
LIN {X 78.799,Y 65.314,Z 63.659,A 180.000,B 0.000,C 180.000} C_DIS
LIN {X 78.874,Y 65.289,Z 63.656,A 180.000,B 0.000,C 180.000} C_DIS
LIN {X 78.948,Y 65.264,Z 63.654,A 180.000,B 0.000,C 180.000} C_DIS
LIN {X 79.023,Y 65.239,Z 63.651,A 180.000,B 0.000,C 180.000} C_DIS
LIN {X 79.098,Y 65.213,Z 63.648,A 180.000,B 0.000,C 180.000} C_DIS
LIN {X 79.247,Y 65.163,Z 63.643,A 180.000,B 0.000,C 180.000} C_DIS
LIN {X 79.396,Y 65.113,Z 63.639,A 180.000,B 0.000,C 180.000} C_DIS
LIN {X 79.545,Y 65.062,Z 63.634,A 180.000,B 0.000,C 180.000} C_DIS
LIN {X 79.694,Y 65.012,Z 63.629,A 180.000,B 0.000,C 180.000} C_DIS
LIN {X 79.844,Y 64.962,Z 63.624,A 180.000,B 0.000,C 180.000} C_DIS
LIN {X 79.993,Y 64.911,Z 63.620,A 180.000,B 0.000,C 180.000} C_DIS
LIN {X 80.142,Y 64.861,Z 63.615,A 180.000,B 0.000,C 180.000} C_DIS
LIN {X 80.291,Y 64.811,Z 63.610,A 180.000,B 0.000,C 180.000} C_DIS
LIN {X 80.441,Y 64.760,Z 63.606,A 180.000,B 0.000,C 180.000} C_DIS
LIN {X 80.590,Y 64.710,Z 63.602,A 180.000,B 0.000,C 180.000} C_DIS
LIN {X 80.739,Y 64.660,Z 63.597,A 180.000,B 0.000,C 180.000} C_DIS
LIN {X 80.888,Y 64.609,Z 63.593,A 180.000,B 0.000,C 180.000} C_DIS
LIN {X 81.038,Y 64.559,Z 63.589,A 180.000,B 0.000,C 180.000} C_DIS
LIN {X 81.187,Y 64.509,Z 63.585,A 180.000,B 0.000,C 180.000} C_DIS
LIN {X 81.336,Y 64.458,Z 63.581,A 180.000,B 0.000,C 180.000} C_DIS
LIN {X 81.485,Y 64.408,Z 63.577,A 180.000,B 0.000,C 180.000} C_DIS
LIN {X 81.635,Y 64.358,Z 63.573,A 180.000,B 0.000,C 180.000} C_DIS
LIN {X 81.784,Y 64.307,Z 63.570,A 180.000,B 0.000,C 180.000} C_DIS
LIN {X 81.933,Y 64.257,Z 63.566,A 180.000,B 0.000,C 180.000} C_DIS
LIN {X 82.082,Y 64.207,Z 63.562,A 180.000,B 0.000,C 180.000} C_DIS
LIN {X 82.231,Y 64.156,Z 63.559,A 180.000,B 0.000,C 180.000} C_DIS
LIN {X 82.381,Y 64.106,Z 63.556,A 180.000,B 0.000,C 180.000} C_DIS
LIN {X 82.530,Y 64.056,Z 63.552,A 180.000,B 0.000,C 180.000} C_DIS
LIN {X 82.679,Y 64.005,Z 63.549,A 180.000,B 0.000,C 180.000} C_DIS
LIN {X 82.828,Y 63.955,Z 63.546,A 180.000,B 0.000,C 180.000} C_DIS
LIN {X 82.978,Y 63.904,Z 63.543,A 180.000,B 0.000,C 180.000} C_DIS
LIN {X 83.127,Y 63.854,Z 63.540,A 180.000,B 0.000,C 180.000} C_DIS
LIN {X 83.276,Y 63.804,Z 63.537,A 180.000,B 0.000,C 180.000} C_DIS
LIN {X 83.425,Y 63.753,Z 63.534,A 180.000,B 0.000,C 180.000} C_DIS
LIN {X 83.575,Y 63.703,Z 63.532,A 180.000,B 0.000,C 180.000} C_DIS
LIN {X 83.724,Y 63.653,Z 63.529,A 180.000,B 0.000,C 180.000} C_DIS
LIN {X 83.873,Y 63.602,Z 63.527,A 180.000,B 0.000,C 180.000} C_DIS
LIN {X 84.172,Y 63.502,Z 63.522,A 180.000,B 0.000,C 180.000} C_DIS
LIN {X 84.470,Y 63.401,Z 63.518,A 180.000,B 0.000,C 180.000} C_DIS
LIN {X 84.769,Y 63.300,Z 63.514,A 180.000,B 0.000,C 180.000} C_DIS
LIN {X 85.067,Y 63.200,Z 63.511,A 180.000,B 0.000,C 180.000} C_DIS
LIN {X 85.365,Y 63.099,Z 63.508,A 180.000,B 0.000,C 180.000} C_DIS
LIN {X 85.664,Y 62.998,Z 63.505,A 180.000,B 0.000,C 180.000} C_DIS
LIN {X 85.962,Y 62.898,Z 63.503,A 180.000,B 0.000,C 180.000} C_DIS
LIN {X 86.261,Y 62.797,Z 63.502,A 180.000,B 0.000,C 180.000} C_DIS
LIN {X 86.559,Y 62.696,Z 63.501,A 180.000,B 0.000,C 180.000} C_DIS
LIN {X 86.858,Y 62.596,Z 63.500,A 180.000,B 0.000,C 180.000} C_DIS
LIN {X 87.077,Y 62.522,Z 63.500,A 180.000,B 0.000,C 180.000} C_DIS
; Cutting Move Starts
LIN {X 96.464,Y 59.355,Z 63.500,A 180.000,B 0.000,C 180.000} C_DIS
LIN {X 96.539,Y 59.329,Z 63.500,A 180.000,B 0.000,C 180.000} C_DIS
LIN {X 96.718,Y 59.257,Z 63.500,A 180.000,B 0.000,C 180.000} C_DIS
LIN {X 96.897,Y 59.186,Z 63.500,A 180.000,B 0.000,C 180.000} C_DIS
LIN {X 97.075,Y 59.119,Z 63.500,A 180.000,B 0.000,C 180.000} C_DIS
LIN {X 97.254,Y 59.050,Z 63.500,A 180.000,B 0.000,C 180.000} C_DIS
LIN {X 97.374,Y 58.997,Z 63.500,A 180.000,B 0.000,C 180.000} C_DIS
LIN {X 97.790,Y 58.812,Z 63.500,A 180.000,B 0.000,C 180.000} C_DIS
LIN {X 97.969,Y 58.729,Z 63.500,A 180.000,B 0.000,C 180.000} C_DIS
LIN {X 98.141,Y 58.640,Z 63.500,A 180.000,B 0.000,C 180.000} C_DIS
LIN {X 98.505,Y 58.449,Z 63.500,A 180.000,B 0.000,C 180.000} C_DIS
LIN {X 98.684,Y 58.352,Z 63.500,A 180.000,B 0.000,C 180.000} C_DIS
LIN {X 98.799,Y 58.282,Z 63.500,A 180.000,B 0.000,C 180.000} C_DIS
LIN {X 99.221,Y 58.026,Z 63.500,A 180.000,B 0.000,C 180.000} C_DIS
LIN {X 99.378,Y 57.925,Z 63.500,A 180.000,B 0.000,C 180.000} C_DIS
LIN {X 99.892,Y 57.567,Z 63.500,A 180.000,B 0.000,C 180.000} C_DIS
LIN {X 99.936,Y 57.536,Z 63.500,A 180.000,B 0.000,C 180.000} C_DIS
LIN {X 100.114,Y 57.397,Z 63.500,A 180.000,B 0.000,C 180.000} C_DIS
LIN {X 100.472,Y 57.113,Z 63.500,A 180.000,B 0.000,C 180.000} C_DIS
LIN {X 100.573,Y 57.031,Z 63.500,A 180.000,B 0.000,C 180.000} C_DIS
LIN {X 100.651,Y 56.962,Z 63.500,A 180.000,B 0.000,C 180.000} C_DIS
LIN {X 101.008,Y 56.640,Z 63.500,A 180.000,B 0.000,C 180.000} C_DIS
LIN {X 101.167,Y 56.495,Z 63.500,A 180.000,B 0.000,C 180.000} C_DIS
LIN {X 101.187,Y 56.474,Z 63.500,A 180.000,B 0.000,C 180.000} C_DIS
LIN {X 101.342,Y 56.316,Z 63.500,A 180.000,B 0.000,C 180.000} C_DIS
LIN {X 101.545,Y 56.109,Z 63.500,A 180.000,B 0.000,C 180.000} C_DIS
LIN {X 101.691,Y 55.958,Z 63.500,A 180.000,B 0.000,C 180.000} C_DIS
LIN {X 101.723,Y 55.923,Z 63.500,A 180.000,B 0.000,C 180.000} C_DIS
LIN {X 101.847,Y 55.779,Z 63.500,A 180.000,B 0.000,C 180.000} C_DIS
LIN {X 102.155,Y 55.422,Z 63.500,A 180.000,B 0.000,C 180.000} C_DIS
LIN {X 102.260,Y 55.294,Z 63.500,A 180.000,B 0.000,C 180.000} C_DIS
LIN {X 102.617,Y 54.822,Z 63.500,A 180.000,B 0.000,C 180.000} C_DIS
LIN {X 102.702,Y 54.707,Z 63.500,A 180.000,B 0.000,C 180.000} C_DIS
LIN {X 102.796,Y 54.566,Z 63.500,A 180.000,B 0.000,C 180.000} C_DIS
LIN {X 103.058,Y 54.171,Z 63.500,A 180.000,B 0.000,C 180.000} C_DIS
LIN {X 103.153,Y 54.019,Z 63.500,A 180.000,B 0.000,C 180.000} C_DIS
LIN {X 103.169,Y 53.992,Z 63.500,A 180.000,B 0.000,C 180.000} C_DIS
LIN {X 103.375,Y 53.634,Z 63.500,A 180.000,B 0.000,C 180.000} C_DIS
LIN {X 103.478,Y 53.455,Z 63.500,A 180.000,B 0.000,C 180.000} C_DIS
LIN {X 103.511,Y 53.397,Z 63.500,A 180.000,B 0.000,C 180.000} C_DIS
LIN {X 103.572,Y 53.277,Z 63.500,A 180.000,B 0.000,C 180.000} C_DIS
LIN {X 103.749,Y 52.919,Z 63.500,A 180.000,B 0.000,C 180.000} C_DIS
LIN {X 103.838,Y 52.740,Z 63.500,A 180.000,B 0.000,C 180.000} C_DIS
LIN {X 103.869,Y 52.674,Z 63.500,A 180.000,B 0.000,C 180.000} C_DIS
LIN {X 103.916,Y 52.562,Z 63.500,A 180.000,B 0.000,C 180.000} C_DIS
LIN {X 104.066,Y 52.204,Z 63.500,A 180.000,B 0.000,C 180.000} C_DIS
LIN {X 104.141,Y 52.025,Z 63.500,A 180.000,B 0.000,C 180.000} C_DIS
LIN {X 104.208,Y 51.847,Z 63.500,A 180.000,B 0.000,C 180.000} C_DIS
LIN {X 104.394,Y 51.310,Z 63.500,A 180.000,B 0.000,C 180.000} C_DIS
LIN {X 104.405,Y 51.278,Z 63.500,A 180.000,B 0.000,C 180.000} C_DIS
LIN {X 104.449,Y 51.131,Z 63.500,A 180.000,B 0.000,C 180.000} C_DIS
LIN {X 104.599,Y 50.595,Z 63.500,A 180.000,B 0.000,C 180.000} C_DIS
LIN {X 104.645,Y 50.416,Z 63.500,A 180.000,B 0.000,C 180.000} C_DIS
LIN {X 104.683,Y 50.238,Z 63.500,A 180.000,B 0.000,C 180.000} C_DIS
LIN {X 104.762,Y 49.861,Z 63.500,A 180.000,B 0.000,C 180.000} C_DIS
LIN {X 104.795,Y 49.701,Z 63.500,A 180.000,B 0.000,C 180.000} C_DIS
LIN {X 104.822,Y 49.523,Z 63.500,A 180.000,B 0.000,C 180.000} C_DIS
LIN {X 104.875,Y 49.165,Z 63.500,A 180.000,B 0.000,C 180.000} C_DIS
LIN {X 104.901,Y 48.986,Z 63.500,A 180.000,B 0.000,C 180.000} C_DIS
LIN {X 104.920,Y 48.807,Z 63.500,A 180.000,B 0.000,C 180.000} C_DIS
LIN {X 104.965,Y 48.271,Z 63.500,A 180.000,B 0.000,C 180.000} C_DIS
LIN {X 104.976,Y 48.092,Z 63.500,A 180.000,B 0.000,C 180.000} C_DIS
LIN {X 104.980,Y 47.914,Z 63.500,A 180.000,B 0.000,C 180.000} C_DIS
LIN {X 104.987,Y 47.556,Z 63.500,A 180.000,B 0.000,C 180.000} C_DIS
LIN {X 104.990,Y 47.377,Z 63.500,A 180.000,B 0.000,C 180.000} C_DIS
LIN {X 104.984,Y 47.198,Z 63.500,A 180.000,B 0.000,C 180.000} C_DIS
LIN {X 104.961,Y 46.662,Z 63.500,A 180.000,B 0.000,C 180.000} C_DIS
LIN {X 104.948,Y 46.483,Z 63.500,A 180.000,B 0.000,C 180.000} C_DIS
LIN {X 104.891,Y 45.947,Z 63.500,A 180.000,B 0.000,C 180.000} C_DIS
LIN {X 104.870,Y 45.768,Z 63.500,A 180.000,B 0.000,C 180.000} C_DIS
LIN {X 104.840,Y 45.590,Z 63.500,A 180.000,B 0.000,C 180.000} C_DIS
LIN {X 104.762,Y 45.133,Z 63.500,A 180.000,B 0.000,C 180.000} C_DIS
LIN {X 104.748,Y 45.053,Z 63.500,A 180.000,B 0.000,C 180.000} C_DIS
LIN {X 104.709,Y 44.874,Z 63.500,A 180.000,B 0.000,C 180.000} C_DIS
LIN {X 104.583,Y 44.338,Z 63.500,A 180.000,B 0.000,C 180.000} C_DIS
LIN {X 104.534,Y 44.159,Z 63.500,A 180.000,B 0.000,C 180.000} C_DIS
LIN {X 104.372,Y 43.623,Z 63.500,A 180.000,B 0.000,C 180.000} C_DIS
LIN {X 104.313,Y 43.444,Z 63.500,A 180.000,B 0.000,C 180.000} C_DIS
LIN {X 104.246,Y 43.266,Z 63.500,A 180.000,B 0.000,C 180.000} C_DIS
LIN {X 104.113,Y 42.908,Z 63.500,A 180.000,B 0.000,C 180.000} C_DIS
LIN {X 104.047,Y 42.739,Z 63.500,A 180.000,B 0.000,C 180.000} C_DIS
LIN {X 104.043,Y 42.729,Z 63.500,A 180.000,B 0.000,C 180.000} C_DIS
LIN {X 103.964,Y 42.550,Z 63.500,A 180.000,B 0.000,C 180.000} C_DIS
LIN {X 103.804,Y 42.193,Z 63.500,A 180.000,B 0.000,C 180.000} C_DIS
LIN {X 103.721,Y 42.014,Z 63.500,A 180.000,B 0.000,C 180.000} C_DIS
LIN {X 103.690,Y 41.954,Z 63.500,A 180.000,B 0.000,C 180.000} C_DIS
LIN {X 103.440,Y 41.478,Z 63.500,A 180.000,B 0.000,C 180.000} C_DIS
LIN {X 103.342,Y 41.299,Z 63.500,A 180.000,B 0.000,C 180.000} C_DIS
LIN {X 103.332,Y 41.284,Z 63.500,A 180.000,B 0.000,C 180.000} C_DIS
LIN {X 103.016,Y 40.763,Z 63.500,A 180.000,B 0.000,C 180.000} C_DIS
LIN {X 102.975,Y 40.696,Z 63.500,A 180.000,B 0.000,C 180.000} C_DIS
LIN {X 102.899,Y 40.584,Z 63.500,A 180.000,B 0.000,C 180.000} C_DIS
LIN {X 102.617,Y 40.180,Z 63.500,A 180.000,B 0.000,C 180.000} C_DIS
LIN {X 102.524,Y 40.048,Z 63.500,A 180.000,B 0.000,C 180.000} C_DIS
LIN {X 102.438,Y 39.938,Z 63.500,A 180.000,B 0.000,C 180.000} C_DIS
LIN {X 102.100,Y 39.511,Z 63.500,A 180.000,B 0.000,C 180.000} C_DIS
LIN {X 102.081,Y 39.488,Z 63.500,A 180.000,B 0.000,C 180.000} C_DIS
LIN {X 101.947,Y 39.333,Z 63.500,A 180.000,B 0.000,C 180.000} C_DIS
LIN {X 101.625,Y 38.975,Z 63.500,A 180.000,B 0.000,C 180.000} C_DIS
LIN {X 101.545,Y 38.886,Z 63.500,A 180.000,B 0.000,C 180.000} C_DIS
LIN {X 101.458,Y 38.796,Z 63.500,A 180.000,B 0.000,C 180.000} C_DIS
LIN {X 101.008,Y 38.357,Z 63.500,A 180.000,B 0.000,C 180.000} C_DIS
LIN {X 100.904,Y 38.260,Z 63.500,A 180.000,B 0.000,C 180.000} C_DIS
LIN {X 100.829,Y 38.196,Z 63.500,A 180.000,B 0.000,C 180.000} C_DIS
LIN {X 100.472,Y 37.888,Z 63.500,A 180.000,B 0.000,C 180.000} C_DIS
LIN {X 100.293,Y 37.740,Z 63.500,A 180.000,B 0.000,C 180.000} C_DIS
LIN {X 99.800,Y 37.366,Z 63.500,A 180.000,B 0.000,C 180.000} C_DIS
LIN {X 99.757,Y 37.334,Z 63.500,A 180.000,B 0.000,C 180.000} C_DIS
LIN {X 99.578,Y 37.212,Z 63.500,A 180.000,B 0.000,C 180.000} C_DIS
LIN {X 99.221,Y 36.975,Z 63.500,A 180.000,B 0.000,C 180.000} C_DIS
LIN {X 99.042,Y 36.860,Z 63.500,A 180.000,B 0.000,C 180.000} C_DIS
LIN {X 98.990,Y 36.830,Z 63.500,A 180.000,B 0.000,C 180.000} C_DIS
LIN {X 98.505,Y 36.550,Z 63.500,A 180.000,B 0.000,C 180.000} C_DIS
LIN {X 98.365,Y 36.472,Z 63.500,A 180.000,B 0.000,C 180.000} C_DIS
LIN {X 98.327,Y 36.453,Z 63.500,A 180.000,B 0.000,C 180.000} C_DIS
LIN {X 97.790,Y 36.187,Z 63.500,A 180.000,B 0.000,C 180.000} C_DIS
LIN {X 97.636,Y 36.115,Z 63.500,A 180.000,B 0.000,C 180.000} C_DIS
LIN {X 97.612,Y 36.105,Z 63.500,A 180.000,B 0.000,C 180.000} C_DIS
LIN {X 97.075,Y 35.880,Z 63.500,A 180.000,B 0.000,C 180.000} C_DIS
LIN {X 96.897,Y 35.810,Z 63.500,A 180.000,B 0.000,C 180.000} C_DIS
LIN {X 96.360,Y 35.623,Z 63.500,A 180.000,B 0.000,C 180.000} C_DIS
LIN {X 96.227,Y 35.578,Z 63.500,A 180.000,B 0.000,C 180.000} C_DIS
LIN {X 96.181,Y 35.565,Z 63.500,A 180.000,B 0.000,C 180.000} C_DIS
LIN {X 96.003,Y 35.515,Z 63.500,A 180.000,B 0.000,C 180.000} C_DIS
LIN {X 95.589,Y 35.400,Z 63.500,A 180.000,B 0.000,C 180.000} C_DIS
LIN {X 95.466,Y 35.367,Z 63.500,A 180.000,B 0.000,C 180.000} C_DIS
LIN {X 95.288,Y 35.328,Z 63.500,A 180.000,B 0.000,C 180.000} C_DIS
LIN {X 94.783,Y 35.221,Z 63.500,A 180.000,B 0.000,C 180.000} C_DIS
LIN {X 94.751,Y 35.214,Z 63.500,A 180.000,B 0.000,C 180.000} C_DIS
LIN {X 94.573,Y 35.185,Z 63.500,A 180.000,B 0.000,C 180.000} C_DIS
LIN {X 94.036,Y 35.106,Z 63.500,A 180.000,B 0.000,C 180.000} C_DIS
LIN {X 93.857,Y 35.084,Z 63.500,A 180.000,B 0.000,C 180.000} C_DIS
LIN {X 93.679,Y 35.069,Z 63.500,A 180.000,B 0.000,C 180.000} C_DIS
LIN {X 93.321,Y 35.040,Z 63.500,A 180.000,B 0.000,C 180.000} C_DIS
LIN {X 93.142,Y 35.026,Z 63.500,A 180.000,B 0.000,C 180.000} C_DIS
LIN {X 92.964,Y 35.021,Z 63.500,A 180.000,B 0.000,C 180.000} C_DIS
LIN {X 92.606,Y 35.014,Z 63.500,A 180.000,B 0.000,C 180.000} C_DIS
LIN {X 92.427,Y 35.010,Z 63.500,A 180.000,B 0.000,C 180.000} C_DIS
LIN {X 92.249,Y 35.014,Z 63.500,A 180.000,B 0.000,C 180.000} C_DIS
LIN {X 91.712,Y 35.037,Z 63.500,A 180.000,B 0.000,C 180.000} C_DIS
LIN {X 91.599,Y 35.042,Z 63.500,A 180.000,B 0.000,C 180.000} C_DIS
LIN {X 91.533,Y 35.047,Z 63.500,A 180.000,B 0.000,C 180.000} C_DIS
LIN {X 91.355,Y 35.066,Z 63.500,A 180.000,B 0.000,C 180.000} C_DIS
LIN {X 90.997,Y 35.104,Z 63.500,A 180.000,B 0.000,C 180.000} C_DIS
LIN {X 90.818,Y 35.123,Z 63.500,A 180.000,B 0.000,C 180.000} C_DIS
LIN {X 90.640,Y 35.152,Z 63.500,A 180.000,B 0.000,C 180.000} C_DIS
LIN {X 90.103,Y 35.243,Z 63.500,A 180.000,B 0.000,C 180.000} C_DIS
LIN {X 89.925,Y 35.279,Z 63.500,A 180.000,B 0.000,C 180.000} C_DIS
LIN {X 89.388,Y 35.406,Z 63.500,A 180.000,B 0.000,C 180.000} C_DIS
LIN {X 89.209,Y 35.451,Z 63.500,A 180.000,B 0.000,C 180.000} C_DIS
LIN {X 89.031,Y 35.505,Z 63.500,A 180.000,B 0.000,C 180.000} C_DIS
LIN {X 88.792,Y 35.577,Z 63.500,A 180.000,B 0.000,C 180.000} C_DIS
LIN {X 88.790,Y 35.578,Z 63.500,A 180.000,B 0.000,C 180.000} C_DIS
LIN {X 88.788,Y 35.578,Z 63.500,A 180.000,B 0.000,C 180.000} C_DIS
LIN {X 88.673,Y 35.605,Z 63.500,A 180.000,B 0.000,C 180.000} C_DIS
LIN {X 88.494,Y 35.659,Z 63.500,A 180.000,B 0.000,C 180.000} C_DIS
LIN {X 45.590,Y 50.133,Z 63.500,A 180.000,B 0.000,C 180.000} C_DIS
LIN {X 45.411,Y 50.194,Z 63.500,A 180.000,B 0.000,C 180.000} C_DIS
LIN {X 45.296,Y 50.238,Z 63.500,A 180.000,B 0.000,C 180.000} C_DIS
LIN {X 45.232,Y 50.265,Z 63.500,A 180.000,B 0.000,C 180.000} C_DIS
LIN {X 45.053,Y 50.353,Z 63.500,A 180.000,B 0.000,C 180.000} C_DIS
LIN {X 44.944,Y 50.416,Z 63.500,A 180.000,B 0.000,C 180.000} C_DIS
LIN {X 44.874,Y 50.461,Z 63.500,A 180.000,B 0.000,C 180.000} C_DIS
LIN {X 44.785,Y 50.522,Z 63.500,A 180.000,B 0.000,C 180.000} C_DIS
LIN {X 44.696,Y 50.590,Z 63.500,A 180.000,B 0.000,C 180.000} C_DIS
LIN {X 44.689,Y 50.595,Z 63.500,A 180.000,B 0.000,C 180.000} C_DIS
LIN {X 44.603,Y 50.667,Z 63.500,A 180.000,B 0.000,C 180.000} C_DIS
LIN {X 44.517,Y 50.746,Z 63.500,A 180.000,B 0.000,C 180.000} C_DIS
LIN {X 44.488,Y 50.774,Z 63.500,A 180.000,B 0.000,C 180.000} C_DIS
LIN {X 44.410,Y 50.855,Z 63.500,A 180.000,B 0.000,C 180.000} C_DIS
LIN {X 44.338,Y 50.936,Z 63.500,A 180.000,B 0.000,C 180.000} C_DIS
LIN {X 44.325,Y 50.953,Z 63.500,A 180.000,B 0.000,C 180.000} C_DIS
LIN {X 44.254,Y 51.042,Z 63.500,A 180.000,B 0.000,C 180.000} C_DIS
LIN {X 44.189,Y 51.131,Z 63.500,A 180.000,B 0.000,C 180.000} C_DIS
LIN {X 44.159,Y 51.176,Z 63.500,A 180.000,B 0.000,C 180.000} C_DIS
LIN {X 44.077,Y 51.310,Z 63.500,A 180.000,B 0.000,C 180.000} C_DIS
LIN {X 43.984,Y 51.489,Z 63.500,A 180.000,B 0.000,C 180.000} C_DIS
LIN {X 43.981,Y 51.497,Z 63.500,A 180.000,B 0.000,C 180.000} C_DIS
LIN {X 43.909,Y 51.668,Z 63.500,A 180.000,B 0.000,C 180.000} C_DIS
LIN {X 43.849,Y 51.847,Z 63.500,A 180.000,B 0.000,C 180.000} C_DIS
LIN {X 43.804,Y 52.025,Z 63.500,A 180.000,B 0.000,C 180.000} C_DIS
LIN {X 43.802,Y 52.035,Z 63.500,A 180.000,B 0.000,C 180.000} C_DIS
LIN {X 43.772,Y 52.204,Z 63.500,A 180.000,B 0.000,C 180.000} C_DIS
LIN {X 43.754,Y 52.383,Z 63.500,A 180.000,B 0.000,C 180.000} C_DIS
LIN {X 43.748,Y 52.562,Z 63.500,A 180.000,B 0.000,C 180.000} C_DIS
LIN {X 43.756,Y 52.740,Z 63.500,A 180.000,B 0.000,C 180.000} C_DIS
LIN {X 43.776,Y 52.919,Z 63.500,A 180.000,B 0.000,C 180.000} C_DIS
LIN {X 43.802,Y 53.064,Z 63.500,A 180.000,B 0.000,C 180.000} C_DIS
LIN {X 43.809,Y 53.098,Z 63.500,A 180.000,B 0.000,C 180.000} C_DIS
LIN {X 43.856,Y 53.277,Z 63.500,A 180.000,B 0.000,C 180.000} C_DIS
LIN {X 43.916,Y 53.455,Z 63.500,A 180.000,B 0.000,C 180.000} C_DIS
LIN {X 50.248,Y 72.226,Z 63.500,A 180.000,B 0.000,C 180.000} C_DIS
LIN {X 50.311,Y 72.405,Z 63.500,A 180.000,B 0.000,C 180.000} C_DIS
LIN {X 50.388,Y 72.584,Z 63.500,A 180.000,B 0.000,C 180.000} C_DIS
LIN {X 50.416,Y 72.640,Z 63.500,A 180.000,B 0.000,C 180.000} C_DIS
LIN {X 50.484,Y 72.763,Z 63.500,A 180.000,B 0.000,C 180.000} C_DIS
LIN {X 50.595,Y 72.936,Z 63.500,A 180.000,B 0.000,C 180.000} C_DIS
LIN {X 50.599,Y 72.941,Z 63.500,A 180.000,B 0.000,C 180.000} C_DIS
LIN {X 50.665,Y 73.031,Z 63.500,A 180.000,B 0.000,C 180.000} C_DIS
LIN {X 50.737,Y 73.120,Z 63.500,A 180.000,B 0.000,C 180.000} C_DIS
LIN {X 50.774,Y 73.162,Z 63.500,A 180.000,B 0.000,C 180.000} C_DIS
LIN {X 50.905,Y 73.299,Z 63.500,A 180.000,B 0.000,C 180.000} C_DIS
LIN {X 50.953,Y 73.343,Z 63.500,A 180.000,B 0.000,C 180.000} C_DIS
LIN {X 51.112,Y 73.478,Z 63.500,A 180.000,B 0.000,C 180.000} C_DIS
LIN {X 51.131,Y 73.493,Z 63.500,A 180.000,B 0.000,C 180.000} C_DIS
LIN {X 51.310,Y 73.616,Z 63.500,A 180.000,B 0.000,C 180.000} C_DIS
LIN {X 51.376,Y 73.656,Z 63.500,A 180.000,B 0.000,C 180.000} C_DIS
LIN {X 51.489,Y 73.719,Z 63.500,A 180.000,B 0.000,C 180.000} C_DIS
LIN {X 51.668,Y 73.803,Z 63.500,A 180.000,B 0.000,C 180.000} C_DIS
LIN {X 51.749,Y 73.835,Z 63.500,A 180.000,B 0.000,C 180.000} C_DIS
LIN {X 51.847,Y 73.870,Z 63.500,A 180.000,B 0.000,C 180.000} C_DIS
LIN {X 52.025,Y 73.923,Z 63.500,A 180.000,B 0.000,C 180.000} C_DIS
LIN {X 52.204,Y 73.961,Z 63.500,A 180.000,B 0.000,C 180.000} C_DIS
LIN {X 52.383,Y 73.987,Z 63.500,A 180.000,B 0.000,C 180.000} C_DIS
LIN {X 52.562,Y 73.999,Z 63.500,A 180.000,B 0.000,C 180.000} C_DIS
LIN {X 52.740,Y 73.998,Z 63.500,A 180.000,B 0.000,C 180.000} C_DIS
LIN {X 52.919,Y 73.985,Z 63.500,A 180.000,B 0.000,C 180.000} C_DIS
LIN {X 53.098,Y 73.958,Z 63.500,A 180.000,B 0.000,C 180.000} C_DIS
LIN {X 53.277,Y 73.918,Z 63.500,A 180.000,B 0.000,C 180.000} C_DIS
LIN {X 53.455,Y 73.864,Z 63.500,A 180.000,B 0.000,C 180.000} C_DIS
LIN {X 83.198,Y 63.830,Z 63.500,A 180.000,B 0.000,C 180.000} C_DIS
LIN {X 87.077,Y 62.522,Z 63.500,A 180.000,B 0.000,C 180.000} C_DIS
; Link Move Starts
LIN {X 87.375,Y 62.421,Z 63.500,A 180.000,B 0.000,C 180.000} C_DIS
LIN {X 87.674,Y 62.320,Z 63.499,A 180.000,B 0.000,C 180.000} C_DIS
LIN {X 87.972,Y 62.220,Z 63.498,A 180.000,B 0.000,C 180.000} C_DIS
LIN {X 88.270,Y 62.119,Z 63.496,A 180.000,B 0.000,C 180.000} C_DIS
LIN {X 88.569,Y 62.018,Z 63.494,A 180.000,B 0.000,C 180.000} C_DIS
LIN {X 88.867,Y 61.918,Z 63.491,A 180.000,B 0.000,C 180.000} C_DIS
LIN {X 89.166,Y 61.817,Z 63.488,A 180.000,B 0.000,C 180.000} C_DIS
LIN {X 89.464,Y 61.716,Z 63.485,A 180.000,B 0.000,C 180.000} C_DIS
LIN {X 89.763,Y 61.615,Z 63.481,A 180.000,B 0.000,C 180.000} C_DIS
LIN {X 90.061,Y 61.515,Z 63.477,A 180.000,B 0.000,C 180.000} C_DIS
LIN {X 90.360,Y 61.414,Z 63.472,A 180.000,B 0.000,C 180.000} C_DIS
LIN {X 90.509,Y 61.364,Z 63.469,A 180.000,B 0.000,C 180.000} C_DIS
LIN {X 90.658,Y 61.313,Z 63.467,A 180.000,B 0.000,C 180.000} C_DIS
LIN {X 90.807,Y 61.263,Z 63.464,A 180.000,B 0.000,C 180.000} C_DIS
LIN {X 90.957,Y 61.213,Z 63.461,A 180.000,B 0.000,C 180.000} C_DIS
LIN {X 91.106,Y 61.162,Z 63.459,A 180.000,B 0.000,C 180.000} C_DIS
LIN {X 91.255,Y 61.112,Z 63.456,A 180.000,B 0.000,C 180.000} C_DIS
LIN {X 91.404,Y 61.062,Z 63.452,A 180.000,B 0.000,C 180.000} C_DIS
LIN {X 91.554,Y 61.011,Z 63.449,A 180.000,B 0.000,C 180.000} C_DIS
LIN {X 91.703,Y 60.961,Z 63.446,A 180.000,B 0.000,C 180.000} C_DIS
LIN {X 91.852,Y 60.911,Z 63.443,A 180.000,B 0.000,C 180.000} C_DIS
LIN {X 92.001,Y 60.860,Z 63.439,A 180.000,B 0.000,C 180.000} C_DIS
LIN {X 92.151,Y 60.810,Z 63.436,A 180.000,B 0.000,C 180.000} C_DIS
LIN {X 92.300,Y 60.760,Z 63.432,A 180.000,B 0.000,C 180.000} C_DIS
LIN {X 92.449,Y 60.709,Z 63.428,A 180.000,B 0.000,C 180.000} C_DIS
LIN {X 92.598,Y 60.659,Z 63.425,A 180.000,B 0.000,C 180.000} C_DIS
LIN {X 92.748,Y 60.609,Z 63.421,A 180.000,B 0.000,C 180.000} C_DIS
LIN {X 92.897,Y 60.558,Z 63.417,A 180.000,B 0.000,C 180.000} C_DIS
LIN {X 93.046,Y 60.508,Z 63.413,A 180.000,B 0.000,C 180.000} C_DIS
LIN {X 93.195,Y 60.458,Z 63.409,A 180.000,B 0.000,C 180.000} C_DIS
LIN {X 93.345,Y 60.407,Z 63.405,A 180.000,B 0.000,C 180.000} C_DIS
LIN {X 93.494,Y 60.357,Z 63.400,A 180.000,B 0.000,C 180.000} C_DIS
LIN {X 93.643,Y 60.307,Z 63.396,A 180.000,B 0.000,C 180.000} C_DIS
LIN {X 93.792,Y 60.256,Z 63.392,A 180.000,B 0.000,C 180.000} C_DIS
LIN {X 93.941,Y 60.206,Z 63.387,A 180.000,B 0.000,C 180.000} C_DIS
LIN {X 94.091,Y 60.155,Z 63.383,A 180.000,B 0.000,C 180.000} C_DIS
LIN {X 94.240,Y 60.105,Z 63.378,A 180.000,B 0.000,C 180.000} C_DIS
LIN {X 94.389,Y 60.055,Z 63.373,A 180.000,B 0.000,C 180.000} C_DIS
LIN {X 94.538,Y 60.004,Z 63.369,A 180.000,B 0.000,C 180.000} C_DIS
LIN {X 94.688,Y 59.954,Z 63.364,A 180.000,B 0.000,C 180.000} C_DIS
LIN {X 94.837,Y 59.904,Z 63.359,A 180.000,B 0.000,C 180.000} C_DIS
LIN {X 94.986,Y 59.853,Z 63.354,A 180.000,B 0.000,C 180.000} C_DIS
LIN {X 95.061,Y 59.828,Z 63.351,A 180.000,B 0.000,C 180.000} C_DIS
LIN {X 95.135,Y 59.803,Z 63.349,A 180.000,B 0.000,C 180.000} C_DIS
LIN {X 95.210,Y 59.778,Z 63.346,A 180.000,B 0.000,C 180.000} C_DIS
LIN {X 95.285,Y 59.753,Z 63.344,A 180.000,B 0.000,C 180.000} C_DIS
LIN {X 95.359,Y 59.728,Z 63.341,A 180.000,B 0.000,C 180.000} C_DIS
LIN {X 95.434,Y 59.702,Z 63.339,A 180.000,B 0.000,C 180.000} C_DIS
LIN {X 95.508,Y 59.677,Z 63.336,A 180.000,B 0.000,C 180.000} C_DIS
LIN {X 95.658,Y 59.627,Z 63.331,A 180.000,B 0.000,C 180.000} C_DIS
LIN {X 95.807,Y 59.577,Z 63.325,A 180.000,B 0.000,C 180.000} C_DIS
LIN {X 95.956,Y 59.526,Z 63.320,A 180.000,B 0.000,C 180.000} C_DIS
LIN {X 96.105,Y 59.476,Z 63.315,A 180.000,B 0.000,C 180.000} C_DIS
LIN {X 96.255,Y 59.425,Z 63.309,A 180.000,B 0.000,C 180.000} C_DIS
LIN {X 96.329,Y 59.400,Z 63.306,A 180.000,B 0.000,C 180.000} C_DIS
LIN {X 96.478,Y 59.350,Z 63.301,A 180.000,B 0.000,C 180.000} C_DIS
LIN {X 96.553,Y 59.324,Z 63.298,A 180.000,B 0.000,C 180.000} C_DIS
LIN {X 96.626,Y 59.296,Z 63.296,A 180.000,B 0.000,C 180.000} C_DIS
LIN {X 96.700,Y 59.268,Z 63.293,A 180.000,B 0.000,C 180.000} C_DIS
LIN {X 96.848,Y 59.213,Z 63.287,A 180.000,B 0.000,C 180.000} C_DIS
LIN {X 96.921,Y 59.185,Z 63.285,A 180.000,B 0.000,C 180.000} C_DIS
LIN {X 97.069,Y 59.131,Z 63.279,A 180.000,B 0.000,C 180.000} C_DIS
LIN {X 97.143,Y 59.103,Z 63.276,A 180.000,B 0.000,C 180.000} C_DIS
LIN {X 97.216,Y 59.075,Z 63.274,A 180.000,B 0.000,C 180.000} C_DIS
LIN {X 97.289,Y 59.045,Z 63.271,A 180.000,B 0.000,C 180.000} C_DIS
LIN {X 97.361,Y 59.013,Z 63.268,A 180.000,B 0.000,C 180.000} C_DIS
LIN {X 97.577,Y 58.917,Z 63.260,A 180.000,B 0.000,C 180.000} C_DIS
LIN {X 97.721,Y 58.853,Z 63.254,A 180.000,B 0.000,C 180.000} C_DIS
LIN {X 97.793,Y 58.821,Z 63.252,A 180.000,B 0.000,C 180.000} C_DIS
LIN {X 97.865,Y 58.789,Z 63.249,A 180.000,B 0.000,C 180.000} C_DIS
LIN {X 97.936,Y 58.756,Z 63.246,A 180.000,B 0.000,C 180.000} C_DIS
LIN {X 98.007,Y 58.721,Z 63.243,A 180.000,B 0.000,C 180.000} C_DIS
LIN {X 98.077,Y 58.684,Z 63.241,A 180.000,B 0.000,C 180.000} C_DIS
LIN {X 98.216,Y 58.611,Z 63.235,A 180.000,B 0.000,C 180.000} C_DIS
LIN {X 98.425,Y 58.502,Z 63.227,A 180.000,B 0.000,C 180.000} C_DIS
LIN {X 98.565,Y 58.429,Z 63.221,A 180.000,B 0.000,C 180.000} C_DIS
LIN {X 98.634,Y 58.391,Z 63.219,A 180.000,B 0.000,C 180.000} C_DIS
LIN {X 98.702,Y 58.352,Z 63.216,A 180.000,B 0.000,C 180.000} C_DIS
LIN {X 98.770,Y 58.311,Z 63.213,A 180.000,B 0.000,C 180.000} C_DIS
LIN {X 99.174,Y 58.066,Z 63.197,A 180.000,B 0.000,C 180.000} C_DIS
LIN {X 99.241,Y 58.025,Z 63.194,A 180.000,B 0.000,C 180.000} C_DIS
LIN {X 99.308,Y 57.983,Z 63.191,A 180.000,B 0.000,C 180.000} C_DIS
LIN {X 99.373,Y 57.940,Z 63.188,A 180.000,B 0.000,C 180.000} C_DIS
LIN {X 99.438,Y 57.895,Z 63.186,A 180.000,B 0.000,C 180.000} C_DIS
LIN {X 99.567,Y 57.805,Z 63.180,A 180.000,B 0.000,C 180.000} C_DIS
LIN {X 99.890,Y 57.580,Z 63.166,A 180.000,B 0.000,C 180.000} C_DIS
LIN {X 99.955,Y 57.534,Z 63.164,A 180.000,B 0.000,C 180.000} C_DIS
LIN {X 100.017,Y 57.486,Z 63.161,A 180.000,B 0.000,C 180.000} C_DIS
LIN {X 100.140,Y 57.388,Z 63.155,A 180.000,B 0.000,C 180.000} C_DIS
LIN {X 100.264,Y 57.290,Z 63.150,A 180.000,B 0.000,C 180.000} C_DIS
LIN {X 100.511,Y 57.094,Z 63.139,A 180.000,B 0.000,C 180.000} C_DIS
LIN {X 100.572,Y 57.045,Z 63.136,A 180.000,B 0.000,C 180.000} C_DIS
LIN {X 100.631,Y 56.993,Z 63.133,A 180.000,B 0.000,C 180.000} C_DIS
LIN {X 100.748,Y 56.887,Z 63.128,A 180.000,B 0.000,C 180.000} C_DIS
LIN {X 101.099,Y 56.571,Z 63.111,A 180.000,B 0.000,C 180.000} C_DIS
LIN {X 101.157,Y 56.517,Z 63.109,A 180.000,B 0.000,C 180.000} C_DIS
LIN {X 101.213,Y 56.462,Z 63.106,A 180.000,B 0.000,C 180.000} C_DIS
LIN {X 101.543,Y 56.124,Z 63.089,A 180.000,B 0.000,C 180.000} C_DIS
LIN {X 101.653,Y 56.012,Z 63.084,A 180.000,B 0.000,C 180.000} C_DIS
LIN {X 101.707,Y 55.954,Z 63.081,A 180.000,B 0.000,C 180.000} C_DIS
LIN {X 101.760,Y 55.896,Z 63.078,A 180.000,B 0.000,C 180.000} C_DIS
LIN {X 102.068,Y 55.538,Z 63.062,A 180.000,B 0.000,C 180.000} C_DIS
LIN {X 102.171,Y 55.418,Z 63.056,A 180.000,B 0.000,C 180.000} C_DIS
LIN {X 102.221,Y 55.358,Z 63.054,A 180.000,B 0.000,C 180.000} C_DIS
LIN {X 102.270,Y 55.296,Z 63.051,A 180.000,B 0.000,C 180.000} C_DIS
LIN {X 102.650,Y 54.794,Z 63.029,A 180.000,B 0.000,C 180.000} C_DIS
LIN {X 102.697,Y 54.730,Z 63.026,A 180.000,B 0.000,C 180.000} C_DIS
LIN {X 102.741,Y 54.665,Z 63.023,A 180.000,B 0.000,C 180.000} C_DIS
LIN {X 103.089,Y 54.140,Z 63.001,A 180.000,B 0.000,C 180.000} C_DIS
LIN {X 103.132,Y 54.074,Z 62.999,A 180.000,B 0.000,C 180.000} C_DIS
LIN {X 103.172,Y 54.006,Z 62.996,A 180.000,B 0.000,C 180.000} C_DIS
LIN {X 103.487,Y 53.460,Z 62.974,A 180.000,B 0.000,C 180.000} C_DIS
LIN {X 103.525,Y 53.391,Z 62.971,A 180.000,B 0.000,C 180.000} C_DIS
LIN {X 103.560,Y 53.321,Z 62.968,A 180.000,B 0.000,C 180.000} C_DIS
LIN {X 103.805,Y 52.827,Z 62.949,A 180.000,B 0.000,C 180.000} C_DIS
LIN {X 103.840,Y 52.757,Z 62.946,A 180.000,B 0.000,C 180.000} C_DIS
LIN {X 103.874,Y 52.685,Z 62.944,A 180.000,B 0.000,C 180.000} C_DIS
LIN {X 103.905,Y 52.613,Z 62.941,A 180.000,B 0.000,C 180.000} C_DIS
LIN {X 104.118,Y 52.105,Z 62.922,A 180.000,B 0.000,C 180.000} C_DIS
LIN {X 104.149,Y 52.032,Z 62.919,A 180.000,B 0.000,C 180.000} C_DIS
LIN {X 104.178,Y 51.959,Z 62.916,A 180.000,B 0.000,C 180.000} C_DIS
LIN {X 104.204,Y 51.885,Z 62.913,A 180.000,B 0.000,C 180.000} C_DIS
LIN {X 104.282,Y 51.662,Z 62.905,A 180.000,B 0.000,C 180.000} C_DIS
LIN {X 104.385,Y 51.364,Z 62.894,A 180.000,B 0.000,C 180.000} C_DIS
LIN {X 104.411,Y 51.290,Z 62.891,A 180.000,B 0.000,C 180.000} C_DIS
LIN {X 104.435,Y 51.215,Z 62.889,A 180.000,B 0.000,C 180.000} C_DIS
LIN {X 104.457,Y 51.139,Z 62.886,A 180.000,B 0.000,C 180.000} C_DIS
LIN {X 104.584,Y 50.684,Z 62.869,A 180.000,B 0.000,C 180.000} C_DIS
LIN {X 104.605,Y 50.608,Z 62.867,A 180.000,B 0.000,C 180.000} C_DIS
LIN {X 104.626,Y 50.532,Z 62.864,A 180.000,B 0.000,C 180.000} C_DIS
LIN {X 104.645,Y 50.456,Z 62.861,A 180.000,B 0.000,C 180.000} C_DIS
LIN {X 104.662,Y 50.379,Z 62.858,A 180.000,B 0.000,C 180.000} C_DIS
LIN {X 104.695,Y 50.225,Z 62.853,A 180.000,B 0.000,C 180.000} C_DIS
LIN {X 104.777,Y 49.840,Z 62.839,A 180.000,B 0.000,C 180.000} C_DIS
LIN {X 104.793,Y 49.763,Z 62.836,A 180.000,B 0.000,C 180.000} C_DIS
LIN {X 104.807,Y 49.685,Z 62.834,A 180.000,B 0.000,C 180.000} C_DIS
LIN {X 104.820,Y 49.607,Z 62.831,A 180.000,B 0.000,C 180.000} C_DIS
LIN {X 104.842,Y 49.452,Z 62.825,A 180.000,B 0.000,C 180.000} C_DIS
LIN {X 104.854,Y 49.374,Z 62.823,A 180.000,B 0.000,C 180.000} C_DIS
LIN {X 104.877,Y 49.218,Z 62.817,A 180.000,B 0.000,C 180.000} C_DIS
LIN {X 104.900,Y 49.062,Z 62.812,A 180.000,B 0.000,C 180.000} C_DIS
LIN {X 104.911,Y 48.984,Z 62.809,A 180.000,B 0.000,C 180.000} C_DIS
LIN {X 104.921,Y 48.906,Z 62.806,A 180.000,B 0.000,C 180.000} C_DIS
LIN {X 104.928,Y 48.827,Z 62.803,A 180.000,B 0.000,C 180.000} C_DIS
LIN {X 104.934,Y 48.749,Z 62.801,A 180.000,B 0.000,C 180.000} C_DIS
LIN {X 104.947,Y 48.592,Z 62.795,A 180.000,B 0.000,C 180.000} C_DIS
LIN {X 104.974,Y 48.278,Z 62.784,A 180.000,B 0.000,C 180.000} C_DIS
LIN {X 104.980,Y 48.200,Z 62.781,A 180.000,B 0.000,C 180.000} C_DIS
LIN {X 104.984,Y 48.121,Z 62.779,A 180.000,B 0.000,C 180.000} C_DIS
LIN {X 104.987,Y 48.042,Z 62.776,A 180.000,B 0.000,C 180.000} C_DIS
LIN {X 104.990,Y 47.885,Z 62.770,A 180.000,B 0.000,C 180.000} C_DIS
LIN {X 104.991,Y 47.806,Z 62.768,A 180.000,B 0.000,C 180.000} C_DIS
LIN {X 104.995,Y 47.649,Z 62.762,A 180.000,B 0.000,C 180.000} C_DIS
LIN {X 104.998,Y 47.491,Z 62.757,A 180.000,B 0.000,C 180.000} C_DIS
LIN {X 104.999,Y 47.412,Z 62.754,A 180.000,B 0.000,C 180.000} C_DIS
LIN {X 104.999,Y 47.334,Z 62.751,A 180.000,B 0.000,C 180.000} C_DIS
LIN {X 104.996,Y 47.255,Z 62.748,A 180.000,B 0.000,C 180.000} C_DIS
LIN {X 104.993,Y 47.176,Z 62.746,A 180.000,B 0.000,C 180.000} C_DIS
LIN {X 104.986,Y 47.019,Z 62.740,A 180.000,B 0.000,C 180.000} C_DIS
LIN {X 104.976,Y 46.783,Z 62.732,A 180.000,B 0.000,C 180.000} C_DIS
LIN {X 104.972,Y 46.704,Z 62.729,A 180.000,B 0.000,C 180.000} C_DIS
LIN {X 104.969,Y 46.625,Z 62.726,A 180.000,B 0.000,C 180.000} C_DIS
LIN {X 104.963,Y 46.547,Z 62.724,A 180.000,B 0.000,C 180.000} C_DIS
LIN {X 104.956,Y 46.469,Z 62.721,A 180.000,B 0.000,C 180.000} C_DIS
LIN {X 104.939,Y 46.312,Z 62.715,A 180.000,B 0.000,C 180.000} C_DIS
LIN {X 104.931,Y 46.234,Z 62.713,A 180.000,B 0.000,C 180.000} C_DIS
LIN {X 104.914,Y 46.077,Z 62.707,A 180.000,B 0.000,C 180.000} C_DIS
LIN {X 104.898,Y 45.920,Z 62.702,A 180.000,B 0.000,C 180.000} C_DIS
LIN {X 104.889,Y 45.842,Z 62.699,A 180.000,B 0.000,C 180.000} C_DIS
LIN {X 104.879,Y 45.764,Z 62.696,A 180.000,B 0.000,C 180.000} C_DIS
LIN {X 104.866,Y 45.686,Z 62.693,A 180.000,B 0.000,C 180.000} C_DIS
LIN {X 104.813,Y 45.376,Z 62.682,A 180.000,B 0.000,C 180.000} C_DIS
LIN {X 104.800,Y 45.298,Z 62.680,A 180.000,B 0.000,C 180.000} C_DIS
LIN {X 104.774,Y 45.143,Z 62.674,A 180.000,B 0.000,C 180.000} C_DIS
LIN {X 104.760,Y 45.065,Z 62.672,A 180.000,B 0.000,C 180.000} C_DIS
LIN {X 104.745,Y 44.988,Z 62.669,A 180.000,B 0.000,C 180.000} C_DIS
LIN {X 104.727,Y 44.911,Z 62.666,A 180.000,B 0.000,C 180.000} C_DIS
LIN {X 104.709,Y 44.835,Z 62.664,A 180.000,B 0.000,C 180.000} C_DIS
LIN {X 104.691,Y 44.758,Z 62.661,A 180.000,B 0.000,C 180.000} C_DIS
LIN {X 104.673,Y 44.681,Z 62.659,A 180.000,B 0.000,C 180.000} C_DIS
LIN {X 104.655,Y 44.605,Z 62.656,A 180.000,B 0.000,C 180.000} C_DIS
LIN {X 104.637,Y 44.528,Z 62.654,A 180.000,B 0.000,C 180.000} C_DIS
LIN {X 104.619,Y 44.451,Z 62.651,A 180.000,B 0.000,C 180.000} C_DIS
LIN {X 104.601,Y 44.375,Z 62.649,A 180.000,B 0.000,C 180.000} C_DIS
LIN {X 104.562,Y 44.222,Z 62.644,A 180.000,B 0.000,C 180.000} C_DIS
LIN {X 104.517,Y 44.071,Z 62.639,A 180.000,B 0.000,C 180.000} C_DIS
LIN {X 104.471,Y 43.920,Z 62.634,A 180.000,B 0.000,C 180.000} C_DIS
LIN {X 104.426,Y 43.770,Z 62.629,A 180.000,B 0.000,C 180.000} C_DIS
LIN {X 104.380,Y 43.619,Z 62.624,A 180.000,B 0.000,C 180.000} C_DIS
LIN {X 104.332,Y 43.469,Z 62.620,A 180.000,B 0.000,C 180.000} C_DIS
LIN {X 104.277,Y 43.321,Z 62.615,A 180.000,B 0.000,C 180.000} C_DIS
